LIN {X 0,Y 312.068,Z 552.76,A -85,B 0,C 180,E1 -16415.031,E2 -16415.031} C_VEL
LIN {X 0,Y 304.932,Z 536.125,A -85,B 0,C 180,E1 -16417.056,E2 -16417.056} C_VEL
LIN {X 0,Y 298.517,Z 522.21,A -85,B 0,C 180,E1 -16418.657,E2 -16418.657} C_VEL
LIN {X 0,Y 298.42,Z 521.626,A -85,B 0,C 180,E1 -16418.707,E2 -16418.707} C_VEL
LIN {X 0,Y 298.405,Z 521.628,A -85,B 0,C 180,E1 -16423.103,E2 -16423.103} C_VEL
LIN {X 0,Y 298.409,Z 521.626,A -85,B 0,C 180,E1 -16426.921,E2 -16426.921} C_VEL
LIN {X 0,Y 298.421,Z 521.626,A -85,B 0,C 180,E1 -16431.003,E2 -16431.003} C_VEL
LIN {X 0,Y 298.435,Z 521.723,A -85,B 0,C 180,E1 -16434.866,E2 -16434.866} C_VEL
LIN {X 0,Y 299.612,Z 527.188,A -85,B 0,C 180,E1 -16438.931,E2 -16438.931} C_VEL
LIN {X 0,Y 300.508,Z 532.409,A -85,B 0,C 180,E1 -16442.713,E2 -16442.713} C_VEL
LIN {X 0,Y 300.68,Z 534.35,A -85,B 0,C 180,E1 -16443.977,E2 -16443.977} C_VEL
LIN {X 0,Y 302.293,Z 537.797,A -85,B 0,C 180,E1 -16444.308,E2 -16444.308} C_VEL
LIN {X 0,Y 309.274,Z 552.419,A -85,B 0,C 180,E1 -16445.757,E2 -16445.757} C_VEL
LIN {X 0,Y 315.209,Z 567.429,A -85,B 0,C 180,E1 -16447.268,E2 -16447.268} C_VEL
LIN {X 0,Y 319.843,Z 581.754,A -85,B 0,C 180,E1 -16448.771,E2 -16448.771} C_VEL
LIN {X 0,Y 323.38,Z 594.422,A -85,B 0,C 180,E1 -16450.193,E2 -16450.193} C_VEL
LIN {X 0,Y 321.224,Z 608.572,A -85,B 0,C 180,E1 -16451.337,E2 -16451.337} C_VEL
LIN {X 0,Y 318.47,Z 623.738,A -85,B 0,C 180,E1 -16452.832,E2 -16452.832} C_VEL
LIN {X 0,Y 315.594,Z 637.637,A -85,B 0,C 180,E1 -16454.499,E2 -16454.499} C_VEL
LIN {X 0,Y 312.662,Z 650.484,A -85,B 0,C 180,E1 -16456.347,E2 -16456.347} C_VEL
LIN {X 0,Y 309.659,Z 663.096,A -85,B 0,C 180,E1 -16458.544,E2 -16458.544} C_VEL
LIN {X 0,Y 306.911,Z 673.805,A -85,B 0,C 180,E1 -16460.775,E2 -16460.775} C_VEL
LIN {X 0,Y 304.203,Z 684.215,A -85,B 0,C 180,E1 -16463.365,E2 -16463.365} C_VEL
LIN {X 0,Y 301.918,Z 692.982,A -85,B 0,C 180,E1 -16465.994,E2 -16465.994} C_VEL
LIN {X 0,Y 300.231,Z 700.324,A -85,B 0,C 180,E1 -16468.657,E2 -16468.657} C_VEL
LIN {X 0,Y 298.834,Z 706.332,A -85,B 0,C 180,E1 -16471.346,E2 -16471.346} C_VEL
LIN {X 0,Y 297.932,Z 711.223,A -85,B 0,C 180,E1 -16474.057,E2 -16474.057} C_VEL
LIN {X 0,Y 297.263,Z 715.069,A -85,B 0,C 180,E1 -16476.787,E2 -16476.787} C_VEL
LIN {X 0,Y 296.813,Z 717.858,A -85,B 0,C 180,E1 -16479.539,E2 -16479.539} C_VEL
LIN {X 0,Y 296.638,Z 719.722,A -85,B 0,C 180,E1 -16482.31,E2 -16482.31} C_VEL
LIN {X 0,Y 296.528,Z 720.531,A -85,B 0,C 180,E1 -16485.111,E2 -16485.111} C_VEL
LIN {X 0,Y 296.624,Z 720.427,A -85,B 0,C 180,E1 -16487.938,E2 -16487.938} C_VEL
LIN {X 0,Y 296.912,Z 719.249,A -85,B 0,C 180,E1 -16490.795,E2 -16490.795} C_VEL
LIN {X 0,Y 297.493,Z 717.043,A -85,B 0,C 180,E1 -16493.677,E2 -16493.677} C_VEL
LIN {X 0,Y 298.46,Z 713.748,A -85,B 0,C 180,E1 -16496.575,E2 -16496.575} C_VEL
LIN {X 0,Y 299.949,Z 708.491,A -85,B 0,C 180,E1 -16499.894,E2 -16499.894} C_VEL
LIN {X 0,Y 301.5,Z 703.345,A -85,B 0,C 180,E1 -16502.419,E2 -16502.419} C_VEL
LIN {X 0,Y 303.896,Z 696.084,A -85,B 0,C 180,E1 -16505.319,E2 -16505.319} C_VEL
LIN {X 0,Y 306.912,Z 687.177,A -85,B 0,C 180,E1 -16508.188,E2 -16508.188} C_VEL
LIN {X 0,Y 310.064,Z 677.773,A -85,B 0,C 180,E1 -16510.664,E2 -16510.664} C_VEL
LIN {X 0,Y 313.119,Z 668.301,A -85,B 0,C 180,E1 -16512.76,E2 -16512.76} C_VEL
LIN {X 0,Y 316.594,Z 657.264,A -85,B 0,C 180,E1 -16514.828,E2 -16514.828} C_VEL
LIN {X 0,Y 320.119,Z 645.238,A -85,B 0,C 180,E1 -16516.715,E2 -16516.715} C_VEL
LIN {X 0,Y 323.381,Z 632.92,A -85,B 0,C 180,E1 -16518.334,E2 -16518.334} C_VEL
LIN {X 0,Y 326.636,Z 619.578,A -85,B 0,C 180,E1 -16519.797,E2 -16519.797} C_VEL
LIN {X 0,Y 329.546,Z 605.586,A -85,B 0,C 180,E1 -16521.08,E2 -16521.08} C_VEL
LIN {X 0,Y 330.671,Z 599.403,A -85,B 0,C 180,E1 -16521.561,E2 -16521.561} C_VEL
LIN {X 0,Y 327.161,Z 585.978,A -85,B 0,C 180,E1 -16523.407,E2 -16523.407} C_VEL
LIN {X 0,Y 322.679,Z 573.581,A -85,B 0,C 180,E1 -16525.181,E2 -16525.181} C_VEL
LIN {X 0,Y 318.133,Z 563.085,A -85,B 0,C 180,E1 -16526.729,E2 -16526.729} C_VEL
LIN {X 0,Y 316.669,Z 560.38,A -85,B 0,C 180,E1 -16527.164,E2 -16527.164} C_VEL
LIN {X 0,Y 313.744,Z 557.363,A -85,B 0,C 180,E1 -16527.921,E2 -16527.921} C_VEL
LIN {X 0,Y 304.855,Z 551.294,A -85,B 0,C 180,E1 -16530.139,E2 -16530.139} C_VEL
LIN {X 0,Y 302.177,Z 547.886,A -85,B 0,C 180,E1 -16530.919,E2 -16530.919} C_VEL
LIN {X 0,Y 299.012,Z 543.525,A -85,B 0,C 180,E1 -16531.864,E2 -16531.864} C_VEL
LIN {X 0,Y 298.209,Z 542.203,A -85,B 0,C 180,E1 -16532.117,E2 -16532.117} C_VEL
LIN {X 0,Y 295.75,Z 539.263,A -85,B 0,C 180,E1 -16532.863,E2 -16532.863} C_VEL
LIN {X 0,Y 294.81,Z 537.165,A -85,B 0,C 180,E1 -16533.258,E2 -16533.258} C_VEL
LIN {X 0,Y 294.299,Z 534.199,A -85,B 0,C 180,E1 -16536.048,E2 -16536.048} C_VEL
LIN {X 0,Y 293.364,Z 529.878,A -85,B 0,C 180,E1 -16540.403,E2 -16540.403} C_VEL
LIN {X 0,Y 292.376,Z 525.78,A -85,B 0,C 180,E1 -16544.667,E2 -16544.667} C_VEL
LIN {X 0,Y 291.664,Z 523.407,A -85,B 0,C 180,E1 -16547.474,E2 -16547.474} C_VEL
LIN {X 0,Y 291.529,Z 522.475,A -85,B 0,C 180,E1 -16548.88,E2 -16548.88} C_VEL
LIN {X 0,Y 291.7,Z 522.453,A -85,B 0,C 180,E1 -16551.688,E2 -16551.688} C_VEL
LIN {X 0,Y 291.625,Z 522.464,A -85,B 0,C 180,E1 -16554.468,E2 -16554.468} C_VEL
LIN {X 0,Y 291.884,Z 522.428,A -85,B 0,C 180,E1 -16558.62,E2 -16558.62} C_VEL
LIN {X 0,Y 291.881,Z 522.429,A -85,B 0,C 180,E1 -16561.379,E2 -16561.379} C_VEL
LIN {X 0,Y 291.736,Z 522.455,A -85,B 0,C 180,E1 -16566.918,E2 -16566.918} C_VEL
LIN {X 0,Y 291.619,Z 522.46,A -85,B 0,C 180,E1 -16569.712,E2 -16569.712} C_VEL
LIN {X 0,Y 291.512,Z 522.483,A -85,B 0,C 180,E1 -16573.95,E2 -16573.95} C_VEL
LIN {X 0,Y 291.477,Z 522.439,A -85,B 0,C 180,E1 -16576.818,E2 -16576.818} C_VEL
LIN {X 0,Y 291.485,Z 522.46,A -85,B 0,C 180,E1 -16579.9,E2 -16579.9} C_VEL
LIN {X 0,Y 291.427,Z 522.446,A -85,B 0,C 180,E1 -16584.202,E2 -16584.202} C_VEL
LIN {X 0,Y 291.416,Z 522.525,A -85,B 0,C 180,E1 -16588.247,E2 -16588.247} C_VEL
LIN {X 0,Y 292.765,Z 528.915,A -85,B 0,C 180,E1 -16591.878,E2 -16591.878} C_VEL
LIN {X 0,Y 294.332,Z 536.056,A -85,B 0,C 180,E1 -16595.727,E2 -16595.727} C_VEL
LIN {X 0,Y 296.072,Z 544.172,A -85,B 0,C 180,E1 -16599.859,E2 -16599.859} C_VEL
LIN {X 0,Y 296.764,Z 547.425,A -85,B 0,C 180,E1 -16601.392,E2 -16601.392} C_VEL
LIN {X 0,Y 298.476,Z 553.641,A -85,B 0,C 180,E1 -16603.297,E2 -16603.297} C_VEL
LIN {X 0,Y 301.646,Z 559.124,A -85,B 0,C 180,E1 -16604.262,E2 -16604.262} C_VEL
LIN {X 0,Y 304.024,Z 563.851,A -85,B 0,C 180,E1 -16604.983,E2 -16604.983} C_VEL
LIN {X 0,Y 305.199,Z 565.983,A -85,B 0,C 180,E1 -16605.323,E2 -16605.323} C_VEL
LIN {X 0,Y 307.57,Z 571.571,A -85,B 0,C 180,E1 -16606.035,E2 -16606.035} C_VEL
LIN {X 0,Y 311.717,Z 584.767,A -85,B 0,C 180,E1 -16607.465,E2 -16607.465} C_VEL
LIN {X 0,Y 315.605,Z 601.039,A -85,B 0,C 180,E1 -16609.161,E2 -16609.161} C_VEL
LIN {X 0,Y 317.351,Z 612.191,A -85,B 0,C 180,E1 -16610.314,E2 -16610.314} C_VEL
LIN {X 0,Y 318.943,Z 628.691,A -85,B 0,C 180,E1 -16612.07,E2 -16612.07} C_VEL
LIN {X 0,Y 319.473,Z 641.632,A -85,B 0,C 180,E1 -16613.563,E2 -16613.563} C_VEL
LIN {X 0,Y 316.619,Z 654.375,A -85,B 0,C 180,E1 -16614.754,E2 -16614.754} C_VEL
LIN {X 0,Y 312.952,Z 668.352,A -85,B 0,C 180,E1 -16616.318,E2 -16616.318} C_VEL
LIN {X 0,Y 309.249,Z 681.452,A -85,B 0,C 180,E1 -16618.106,E2 -16618.106} C_VEL
LIN {X 0,Y 305.844,Z 693.144,A -85,B 0,C 180,E1 -16620.016,E2 -16620.016} C_VEL
LIN {X 0,Y 302.262,Z 704.878,A -85,B 0,C 180,E1 -16622.29,E2 -16622.29} C_VEL
LIN {X 0,Y 298.722,Z 716.22,A -85,B 0,C 180,E1 -16624.947,E2 -16624.947} C_VEL
LIN {X 0,Y 295.836,Z 725.738,A -85,B 0,C 180,E1 -16627.662,E2 -16627.662} C_VEL
LIN {X 0,Y 293.626,Z 733.778,A -85,B 0,C 180,E1 -16630.424,E2 -16630.424} C_VEL
LIN {X 0,Y 291.89,Z 740.531,A -85,B 0,C 180,E1 -16633.208,E2 -16633.208} C_VEL
LIN {X 0,Y 290.786,Z 746.03,A -85,B 0,C 180,E1 -16636.015,E2 -16636.015} C_VEL
LIN {X 0,Y 289.975,Z 750.428,A -85,B 0,C 180,E1 -16638.822,E2 -16638.822} C_VEL
LIN {X 0,Y 289.701,Z 753.787,A -85,B 0,C 180,E1 -16641.632,E2 -16641.632} C_VEL
LIN {X 0,Y 289.689,Z 756.102,A -85,B 0,C 180,E1 -16644.433,E2 -16644.433} C_VEL
LIN {X 0,Y 289.668,Z 757.442,A -85,B 0,C 180,E1 -16647.22,E2 -16647.22} C_VEL
LIN {X 0,Y 289.918,Z 757.758,A -85,B 0,C 180,E1 -16650.001,E2 -16650.001} C_VEL
LIN {X 0,Y 289.714,Z 757.082,A -85,B 0,C 180,E1 -16652.782,E2 -16652.782} C_VEL
LIN {X 0,Y 289.791,Z 754.905,A -85,B 0,C 180,E1 -16656.109,E2 -16656.109} C_VEL
LIN {X 0,Y 289.737,Z 752.618,A -85,B 0,C 180,E1 -16658.37,E2 -16658.37} C_VEL
LIN {X 0,Y 290.022,Z 748.721,A -85,B 0,C 180,E1 -16661.18,E2 -16661.18} C_VEL
LIN {X 0,Y 290.777,Z 743.764,A -85,B 0,C 180,E1 -16663.988,E2 -16663.988} C_VEL
LIN {X 0,Y 291.83,Z 737.527,A -85,B 0,C 180,E1 -16666.799,E2 -16666.799} C_VEL
LIN {X 0,Y 293.456,Z 729.927,A -85,B 0,C 180,E1 -16669.591,E2 -16669.591} C_VEL
LIN {X 0,Y 295.573,Z 720.817,A -85,B 0,C 180,E1 -16672.362,E2 -16672.362} C_VEL
LIN {X 0,Y 297.926,Z 711.447,A -85,B 0,C 180,E1 -16674.755,E2 -16674.755} C_VEL
LIN {X 0,Y 300.744,Z 701.517,A -85,B 0,C 180,E1 -16677.032,E2 -16677.032} C_VEL
LIN {X 0,Y 305.458,Z 687.681,A -85,B 0,C 180,E1 -16680.029,E2 -16680.029} C_VEL
LIN {X 0,Y 310.418,Z 674.005,A -85,B 0,C 180,E1 -16682.529,E2 -16682.529} C_VEL
LIN {X 0,Y 315.731,Z 659.951,A -85,B 0,C 180,E1 -16684.721,E2 -16684.721} C_VEL
LIN {X 0,Y 321.64,Z 644.618,A -85,B 0,C 180,E1 -16686.739,E2 -16686.739} C_VEL
LIN {X 0,Y 325.443,Z 627.689,A -85,B 0,C 180,E1 -16689.374,E2 -16689.374} C_VEL
LIN {X 0,Y 327.711,Z 618.124,A -85,B 0,C 180,E1 -16690.865,E2 -16690.865} C_VEL
LIN {X 0,Y 329.683,Z 608.688,A -85,B 0,C 180,E1 -16692.588,E2 -16692.588} C_VEL
LIN {X 0,Y 331.116,Z 602.16,A -85,B 0,C 180,E1 -16694.019,E2 -16694.019} C_VEL
LIN {X 0,Y 332.458,Z 596.698,A -85,B 0,C 180,E1 -16695.485,E2 -16695.485} C_VEL
LIN {X 0,Y 332.805,Z 595.493,A -85,B 0,C 180,E1 -16695.89,E2 -16695.89} C_VEL
LIN {X 0,Y 333.507,Z 593.023,A -85,B 0,C 180,E1 -16697.525,E2 -16697.525} C_VEL
LIN {X 0,Y 334.572,Z 592.021,A -85,B 0,C 180,E1 -16699.37,E2 -16699.37} C_VEL
LIN {X 0,Y 335.825,Z 592.61,A -85,B 0,C 180,E1 -16701.111,E2 -16701.111} C_VEL
LIN {X 0,Y 336.55,Z 593.309,A -85,B 0,C 180,E1 -16701.936,E2 -16701.936} C_VEL
LIN {X 0,Y 336.702,Z 594.466,A -85,B 0,C 180,E1 -16702.423,E2 -16702.423} C_VEL
LIN {X 0,Y 330.299,Z 609.275,A -85,B 0,C 180,E1 -16704.284,E2 -16704.284} C_VEL
LIN {X 0,Y 324.025,Z 623.317,A -85,B 0,C 180,E1 -16706.422,E2 -16706.422} C_VEL
LIN {X 0,Y 318.154,Z 636.055,A -85,B 0,C 180,E1 -16708.728,E2 -16708.728} C_VEL
LIN {X 0,Y 312.432,Z 648.32,A -85,B 0,C 180,E1 -16711.427,E2 -16711.427} C_VEL
LIN {X 0,Y 307.401,Z 658.917,A -85,B 0,C 180,E1 -16714.254,E2 -16714.254} C_VEL
LIN {X 0,Y 303.567,Z 666.914,A -85,B 0,C 180,E1 -16716.824,E2 -16716.824} C_VEL
LIN {X 0,Y 299.75,Z 674.929,A -85,B 0,C 180,E1 -16720.006,E2 -16720.006} C_VEL
LIN {X 0,Y 296.503,Z 681.705,A -85,B 0,C 180,E1 -16723.476,E2 -16723.476} C_VEL
LIN {X 0,Y 294.578,Z 685.761,A -85,B 0,C 180,E1 -16726.198,E2 -16726.198} C_VEL
LIN {X 0,Y 293.106,Z 688.796,A -85,B 0,C 180,E1 -16728.942,E2 -16728.942} C_VEL
LIN {X 0,Y 292.113,Z 690.843,A -85,B 0,C 180,E1 -16731.701,E2 -16731.701} C_VEL
LIN {X 0,Y 291.314,Z 691.996,A -85,B 0,C 180,E1 -16734.463,E2 -16734.463} C_VEL
LIN {X 0,Y 290.669,Z 692.161,A -85,B 0,C 180,E1 -16737.229,E2 -16737.229} C_VEL
LIN {X 0,Y 290.401,Z 691.421,A -85,B 0,C 180,E1 -16740.001,E2 -16740.001} C_VEL
LIN {X 0,Y 290.627,Z 689.591,A -85,B 0,C 180,E1 -16742.773,E2 -16742.773} C_VEL
LIN {X 0,Y 290.747,Z 686.851,A -85,B 0,C 180,E1 -16745.549,E2 -16745.549} C_VEL
LIN {X 0,Y 291.059,Z 683.042,A -85,B 0,C 180,E1 -16748.331,E2 -16748.331} C_VEL
LIN {X 0,Y 291.608,Z 678.11,A -85,B 0,C 180,E1 -16751.117,E2 -16751.117} C_VEL
LIN {X 0,Y 292.432,Z 672.021,A -85,B 0,C 180,E1 -16753.907,E2 -16753.907} C_VEL
LIN {X 0,Y 293.802,Z 664.583,A -85,B 0,C 180,E1 -16756.682,E2 -16756.682} C_VEL
LIN {X 0,Y 295.511,Z 655.655,A -85,B 0,C 180,E1 -16759.449,E2 -16759.449} C_VEL
LIN {X 0,Y 297.707,Z 645.056,A -85,B 0,C 180,E1 -16762.193,E2 -16762.193} C_VEL
LIN {X 0,Y 299.852,Z 634.147,A -85,B 0,C 180,E1 -16764.585,E2 -16764.585} C_VEL
LIN {X 0,Y 302.572,Z 621.424,A -85,B 0,C 180,E1 -16766.933,E2 -16766.933} C_VEL
LIN {X 0,Y 305.365,Z 607.68,A -85,B 0,C 180,E1 -16769.072,E2 -16769.072} C_VEL
LIN {X 0,Y 308.055,Z 593.873,A -85,B 0,C 180,E1 -16770.886,E2 -16770.886} C_VEL
LIN {X 0,Y 310.71,Z 579.23,A -85,B 0,C 180,E1 -16772.494,E2 -16772.494} C_VEL
LIN {X 0,Y 311.817,Z 571.97,A -85,B 0,C 180,E1 -16773.2,E2 -16773.2} C_VEL
LIN {X 0,Y 307.355,Z 559.617,A -85,B 0,C 180,E1 -16774.866,E2 -16774.866} C_VEL
LIN {X 0,Y 301.48,Z 545.18,A -85,B 0,C 180,E1 -16776.741,E2 -16776.741} C_VEL
LIN {X 0,Y 294.433,Z 529.331,A -85,B 0,C 180,E1 -16778.684,E2 -16778.684} C_VEL
LIN {X 0,Y 291.532,Z 523.367,A -85,B 0,C 180,E1 -16779.385,E2 -16779.385} C_VEL
LIN {X 0,Y 291.393,Z 522.501,A -85,B 0,C 180,E1 -16779.483,E2 -16779.483} C_VEL
LIN {X 0,Y 291.315,Z 522.51,A -85,B 0,C 180,E1 -16783.633,E2 -16783.633} C_VEL
LIN {X 0,Y 291.326,Z 522.511,A -85,B 0,C 180,E1 -16787.507,E2 -16787.507} C_VEL
LIN {X 0,Y 291.37,Z 522.505,A -85,B 0,C 180,E1 -16791.16,E2 -16791.16} C_VEL
LIN {X 0,Y 291.399,Z 522.611,A -85,B 0,C 180,E1 -16793.992,E2 -16793.992} C_VEL
LIN {X 0,Y 292.323,Z 526.946,A -85,B 0,C 180,E1 -16797.297,E2 -16797.297} C_VEL
LIN {X 0,Y 293.165,Z 531.342,A -85,B 0,C 180,E1 -16800.563,E2 -16800.563} C_VEL
LIN {X 0,Y 293.678,Z 534.633,A -85,B 0,C 180,E1 -16802.954,E2 -16802.954} C_VEL
LIN {X 0,Y 295.034,Z 537.774,A -85,B 0,C 180,E1 -16803.255,E2 -16803.255} C_VEL
LIN {X 0,Y 297.979,Z 543.093,A -85,B 0,C 180,E1 -16803.852,E2 -16803.852} C_VEL
LIN {X 0,Y 304.245,Z 556.889,A -85,B 0,C 180,E1 -16805.287,E2 -16805.287} C_VEL
LIN {X 0,Y 309.645,Z 570.83,A -85,B 0,C 180,E1 -16806.76,E2 -16806.76} C_VEL
LIN {X 0,Y 314.242,Z 585.645,A -85,B 0,C 180,E1 -16808.394,E2 -16808.394} C_VEL
LIN {X 0,Y 317.025,Z 595.953,A -85,B 0,C 180,E1 -16809.601,E2 -16809.601} C_VEL
LIN {X 0,Y 316.607,Z 600.05,A -85,B 0,C 180,E1 -16809.95,E2 -16809.95} C_VEL
LIN {X 0,Y 314.058,Z 614.736,A -85,B 0,C 180,E1 -16811.234,E2 -16811.234} C_VEL
LIN {X 0,Y 311.281,Z 628.973,A -85,B 0,C 180,E1 -16812.761,E2 -16812.761} C_VEL
LIN {X 0,Y 308.063,Z 643.223,A -85,B 0,C 180,E1 -16814.619,E2 -16814.619} C_VEL
LIN {X 0,Y 304.942,Z 656.155,A -85,B 0,C 180,E1 -16816.674,E2 -16816.674} C_VEL
LIN {X 0,Y 301.888,Z 667.985,A -85,B 0,C 180,E1 -16818.926,E2 -16818.926} C_VEL
LIN {X 0,Y 299.213,Z 678.09,A -85,B 0,C 180,E1 -16821.217,E2 -16821.217} C_VEL
LIN {X 0,Y 296.633,Z 687.902,A -85,B 0,C 180,E1 -16823.878,E2 -16823.878} C_VEL
LIN {X 0,Y 294.416,Z 696.158,A -85,B 0,C 180,E1 -16826.577,E2 -16826.577} C_VEL
LIN {X 0,Y 292.749,Z 702.969,A -85,B 0,C 180,E1 -16829.311,E2 -16829.311} C_VEL
LIN {X 0,Y 291.425,Z 708.624,A -85,B 0,C 180,E1 -16832.072,E2 -16832.072} C_VEL
LIN {X 0,Y 290.624,Z 713.137,A -85,B 0,C 180,E1 -16834.854,E2 -16834.854} C_VEL
LIN {X 0,Y 290.136,Z 715.861,A -85,B 0,C 180,E1 -16836.955,E2 -16836.955} C_VEL
LIN {X 0,Y 289.705,Z 718.53,A -85,B 0,C 180,E1 -16839.775,E2 -16839.775} C_VEL
LIN {X 0,Y 289.528,Z 720.286,A -85,B 0,C 180,E1 -16842.617,E2 -16842.617} C_VEL
LIN {X 0,Y 289.444,Z 721.023,A -85,B 0,C 180,E1 -16845.49,E2 -16845.49} C_VEL
LIN {X 0,Y 289.626,Z 720.652,A -85,B 0,C 180,E1 -16848.848,E2 -16848.848} C_VEL
LIN {X 0,Y 289.907,Z 719.555,A -85,B 0,C 180,E1 -16851.322,E2 -16851.322} C_VEL
LIN {X 0,Y 290.592,Z 717.214,A -85,B 0,C 180,E1 -16854.275,E2 -16854.275} C_VEL
LIN {X 0,Y 291.666,Z 713.805,A -85,B 0,C 180,E1 -16857.245,E2 -16857.245} C_VEL
LIN {X 0,Y 293.125,Z 708.984,A -85,B 0,C 180,E1 -16860.328,E2 -16860.328} C_VEL
LIN {X 0,Y 295.319,Z 702.313,A -85,B 0,C 180,E1 -16863.598,E2 -16863.598} C_VEL
LIN {X 0,Y 297.632,Z 695.728,A -85,B 0,C 180,E1 -16866.178,E2 -16866.178} C_VEL
LIN {X 0,Y 300.896,Z 686.635,A -85,B 0,C 180,E1 -16869.095,E2 -16869.095} C_VEL
LIN {X 0,Y 304.269,Z 677.111,A -85,B 0,C 180,E1 -16871.608,E2 -16871.608} C_VEL
LIN {X 0,Y 308.048,Z 665.732,A -85,B 0,C 180,E1 -16874.092,E2 -16874.092} C_VEL
LIN {X 0,Y 312.114,Z 653.156,A -85,B 0,C 180,E1 -16876.331,E2 -16876.331} C_VEL
LIN {X 0,Y 315.571,Z 641.406,A -85,B 0,C 180,E1 -16878.077,E2 -16878.077} C_VEL
LIN {X 0,Y 319.027,Z 628.425,A -85,B 0,C 180,E1 -16879.706,E2 -16879.706} C_VEL
LIN {X 0,Y 322.493,Z 613.913,A -85,B 0,C 180,E1 -16881.201,E2 -16881.201} C_VEL
LIN {X 0,Y 324.92,Z 602.182,A -85,B 0,C 180,E1 -16882.188,E2 -16882.188} C_VEL
LIN {X 0,Y 323.264,Z 594.426,A -85,B 0,C 180,E1 -16883.283,E2 -16883.283} C_VEL
LIN {X 0,Y 320.154,Z 583.941,A -85,B 0,C 180,E1 -16884.813,E2 -16884.813} C_VEL
LIN {X 0,Y 314.765,Z 570.031,A -85,B 0,C 180,E1 -16886.931,E2 -16886.931} C_VEL
LIN {X 0,Y 309.774,Z 560.044,A -85,B 0,C 180,E1 -16888.593,E2 -16888.593} C_VEL
LIN {X 0,Y 304.543,Z 551.551,A -85,B 0,C 180,E1 -16890.195,E2 -16890.195} C_VEL
LIN {X 0,Y 302.177,Z 547.886,A -85,B 0,C 180,E1 -16890.919,E2 -16890.919} C_VEL
LIN {X 0,Y 300.362,Z 545.843,A -85,B 0,C 180,E1 -16891.451,E2 -16891.451} C_VEL
LIN {X 0,Y 297.343,Z 544.559,A -85,B 0,C 180,E1 -16892.254,E2 -16892.254} C_VEL
LIN {X 0,Y 292.573,Z 543.398,A -85,B 0,C 180,E1 -16893.537,E2 -16893.537} C_VEL
LIN {X 0,Y 290.477,Z 542.015,A -85,B 0,C 180,E1 -16894.169,E2 -16894.169} C_VEL
LIN {X 0,Y 288.354,Z 539.004,A -85,B 0,C 180,E1 -16894.905,E2 -16894.905} C_VEL
LIN {X 0,Y 287.884,Z 537.831,A -85,B 0,C 180,E1 -16895.15,E2 -16895.15} C_VEL
LIN {X 0,Y 287.201,Z 534.564,A -85,B 0,C 180,E1 -16898.465,E2 -16898.465} C_VEL
LIN {X 0,Y 286.6,Z 531.729,A -85,B 0,C 180,E1 -16901.41,E2 -16901.41} C_VEL
LIN {X 0,Y 286.073,Z 529.219,A -85,B 0,C 180,E1 -16904.321,E2 -16904.321} C_VEL
LIN {X 0,Y 285.392,Z 526.753,A -85,B 0,C 180,E1 -16907.194,E2 -16907.194} C_VEL
LIN {X 0,Y 284.654,Z 523.331,A -85,B 0,C 180,E1 -16911.659,E2 -16911.659} C_VEL
LIN {X 0,Y 284.595,Z 523.34,A -85,B 0,C 180,E1 -16914.33,E2 -16914.33} C_VEL
LIN {X 0,Y 284.85,Z 523.304,A -85,B 0,C 180,E1 -16918.586,E2 -16918.586} C_VEL
LIN {X 0,Y 284.847,Z 523.305,A -85,B 0,C 180,E1 -16921.413,E2 -16921.413} C_VEL
LIN {X 0,Y 284.688,Z 523.334,A -85,B 0,C 180,E1 -16927.09,E2 -16927.09} C_VEL
LIN {X 0,Y 284.557,Z 523.342,A -85,B 0,C 180,E1 -16929.955,E2 -16929.955} C_VEL
LIN {X 0,Y 284.468,Z 523.362,A -85,B 0,C 180,E1 -16934.303,E2 -16934.303} C_VEL
LIN {X 0,Y 284.419,Z 523.314,A -85,B 0,C 180,E1 -16937.248,E2 -16937.248} C_VEL
LIN {X 0,Y 284.416,Z 523.348,A -85,B 0,C 180,E1 -16940.239,E2 -16940.239} C_VEL
LIN {X 0,Y 284.386,Z 523.324,A -85,B 0,C 180,E1 -16943.888,E2 -16943.888} C_VEL
LIN {X 0,Y 284.412,Z 523.547,A -85,B 0,C 180,E1 -16947.184,E2 -16947.184} C_VEL
LIN {X 0,Y 284.967,Z 526.134,A -85,B 0,C 180,E1 -16949.148,E2 -16949.148} C_VEL
LIN {X 0,Y 286.625,Z 533.849,A -85,B 0,C 180,E1 -16953.526,E2 -16953.526} C_VEL
LIN {X 0,Y 287.636,Z 538.467,A -85,B 0,C 180,E1 -16955.902,E2 -16955.902} C_VEL
LIN {X 0,Y 290.236,Z 548.399,A -85,B 0,C 180,E1 -16959.917,E2 -16959.917} C_VEL
LIN {X 0,Y 291.625,Z 553.109,A -85,B 0,C 180,E1 -16961.525,E2 -16961.525} C_VEL
LIN {X 0,Y 297.821,Z 563.754,A -85,B 0,C 180,E1 -16963.532,E2 -16963.532} C_VEL
LIN {X 0,Y 300.518,Z 569.122,A -85,B 0,C 180,E1 -16964.378,E2 -16964.378} C_VEL
LIN {X 0,Y 303.271,Z 575.471,A -85,B 0,C 180,E1 -16965.269,E2 -16965.269} C_VEL
LIN {X 0,Y 307.213,Z 588.978,A -85,B 0,C 180,E1 -16966.788,E2 -16966.788} C_VEL
LIN {X 0,Y 310.605,Z 604.754,A -85,B 0,C 180,E1 -16968.529,E2 -16968.529} C_VEL
LIN {X 0,Y 312.093,Z 615.786,A -85,B 0,C 180,E1 -16969.713,E2 -16969.713} C_VEL
LIN {X 0,Y 313.325,Z 632.527,A -85,B 0,C 180,E1 -16971.594,E2 -16971.594} C_VEL
LIN {X 0,Y 313.571,Z 643.992,A -85,B 0,C 180,E1 -16972.964,E2 -16972.964} C_VEL
LIN {X 0,Y 309.745,Z 659.026,A -85,B 0,C 180,E1 -16974.452,E2 -16974.452} C_VEL
LIN {X 0,Y 306.148,Z 671.945,A -85,B 0,C 180,E1 -16976.019,E2 -16976.019} C_VEL
LIN {X 0,Y 302.605,Z 683.749,A -85,B 0,C 180,E1 -16977.714,E2 -16977.714} C_VEL
LIN {X 0,Y 298.55,Z 696.753,A -85,B 0,C 180,E1 -16979.987,E2 -16979.987} C_VEL
LIN {X 0,Y 294.952,Z 707.814,A -85,B 0,C 180,E1 -16982.315,E2 -16982.315} C_VEL
LIN {X 0,Y 291.37,Z 718.597,A -85,B 0,C 180,E1 -16985.034,E2 -16985.034} C_VEL
LIN {X 0,Y 288.404,Z 728.142,A -85,B 0,C 180,E1 -16987.969,E2 -16987.969} C_VEL
LIN {X 0,Y 286.318,Z 735.393,A -85,B 0,C 180,E1 -16990.65,E2 -16990.65} C_VEL
LIN {X 0,Y 284.36,Z 743.165,A -85,B 0,C 180,E1 -16994.226,E2 -16994.226} C_VEL
LIN {X 0,Y 283.146,Z 749.132,A -85,B 0,C 180,E1 -16997.822,E2 -16997.822} C_VEL
LIN {X 0,Y 282.612,Z 753.42,A -85,B 0,C 180,E1 -17001.421,E2 -17001.421} C_VEL
LIN {X 0,Y 282.627,Z 755.697,A -85,B 0,C 180,E1 -17004.293,E2 -17004.293} C_VEL
LIN {X 0,Y 282.589,Z 757.018,A -85,B 0,C 180,E1 -17007.15,E2 -17007.15} C_VEL
LIN {X 0,Y 282.831,Z 757.297,A -85,B 0,C 180,E1 -17010.002,E2 -17010.002} C_VEL
LIN {X 0,Y 282.633,Z 756.603,A -85,B 0,C 180,E1 -17012.852,E2 -17012.852} C_VEL
LIN {X 0,Y 282.7,Z 754.545,A -85,B 0,C 180,E1 -17016.066,E2 -17016.066} C_VEL
LIN {X 0,Y 282.673,Z 752.074,A -85,B 0,C 180,E1 -17018.581,E2 -17018.581} C_VEL
LIN {X 0,Y 283.167,Z 747.036,A -85,B 0,C 180,E1 -17022.18,E2 -17022.18} C_VEL
LIN {X 0,Y 284.075,Z 741.298,A -85,B 0,C 180,E1 -17025.237,E2 -17025.237} C_VEL
LIN {X 0,Y 285.29,Z 735.068,A -85,B 0,C 180,E1 -17027.936,E2 -17027.936} C_VEL
LIN {X 0,Y 287.14,Z 727.116,A -85,B 0,C 180,E1 -17030.789,E2 -17030.789} C_VEL
LIN {X 0,Y 289.52,Z 717.506,A -85,B 0,C 180,E1 -17033.613,E2 -17033.613} C_VEL
LIN {X 0,Y 293.541,Z 704.191,A -85,B 0,C 180,E1 -17037.06,E2 -17037.06} C_VEL
LIN {X 0,Y 298.231,Z 691.414,A -85,B 0,C 180,E1 -17040.052,E2 -17040.052} C_VEL
LIN {X 0,Y 302.45,Z 680.274,A -85,B 0,C 180,E1 -17042.308,E2 -17042.308} C_VEL
LIN {X 0,Y 308.824,Z 664.602,A -85,B 0,C 180,E1 -17044.99,E2 -17044.99} C_VEL
LIN {X 0,Y 315.318,Z 649.165,A -85,B 0,C 180,E1 -17047.2,E2 -17047.2} C_VEL
LIN {X 0,Y 316.584,Z 645.955,A -85,B 0,C 180,E1 -17047.626,E2 -17047.626} C_VEL
LIN {X 0,Y 320.27,Z 632.107,A -85,B 0,C 180,E1 -17049.931,E2 -17049.931} C_VEL
LIN {X 0,Y 322.893,Z 623.265,A -85,B 0,C 180,E1 -17051.338,E2 -17051.338} C_VEL
LIN {X 0,Y 325.265,Z 614.413,A -85,B 0,C 180,E1 -17052.982,E2 -17052.982} C_VEL
LIN {X 0,Y 327.111,Z 607.79,A -85,B 0,C 180,E1 -17054.443,E2 -17054.443} C_VEL
LIN {X 0,Y 329.06,Z 601.713,A -85,B 0,C 180,E1 -17056.131,E2 -17056.131} C_VEL
LIN {X 0,Y 329.641,Z 600.043,A -85,B 0,C 180,E1 -17056.981,E2 -17056.981} C_VEL
LIN {X 0,Y 330.515,Z 598.415,A -85,B 0,C 180,E1 -17058.763,E2 -17058.763} C_VEL
LIN {X 0,Y 331.176,Z 598.203,A -85,B 0,C 180,E1 -17059.816,E2 -17059.816} C_VEL
LIN {X 0,Y 332.414,Z 598.97,A -85,B 0,C 180,E1 -17061.47,E2 -17061.47} C_VEL
LIN {X 0,Y 332.125,Z 600.055,A -85,B 0,C 180,E1 -17061.789,E2 -17061.789} C_VEL
LIN {X 0,Y 325.404,Z 614.025,A -85,B 0,C 180,E1 -17063.662,E2 -17063.662} C_VEL
LIN {X 0,Y 318.875,Z 627.305,A -85,B 0,C 180,E1 -17065.805,E2 -17065.805} C_VEL
LIN {X 0,Y 312.704,Z 639.419,A -85,B 0,C 180,E1 -17068.119,E2 -17068.119} C_VEL
LIN {X 0,Y 307.355,Z 649.865,A -85,B 0,C 180,E1 -17070.516,E2 -17070.516} C_VEL
LIN {X 0,Y 301.951,Z 660.274,A -85,B 0,C 180,E1 -17073.382,E2 -17073.382} C_VEL
LIN {X 0,Y 298.322,Z 667.254,A -85,B 0,C 180,E1 -17075.653,E2 -17075.653} C_VEL
LIN {X 0,Y 294.497,Z 674.593,A -85,B 0,C 180,E1 -17078.548,E2 -17078.548} C_VEL
LIN {X 0,Y 291.109,Z 680.996,A -85,B 0,C 180,E1 -17081.709,E2 -17081.709} C_VEL
LIN {X 0,Y 288.742,Z 685.357,A -85,B 0,C 180,E1 -17084.471,E2 -17084.471} C_VEL
LIN {X 0,Y 286.953,Z 688.77,A -85,B 0,C 180,E1 -17087.267,E2 -17087.267} C_VEL
LIN {X 0,Y 285.677,Z 691.143,A -85,B 0,C 180,E1 -17090.084,E2 -17090.084} C_VEL
LIN {X 0,Y 284.742,Z 692.613,A -85,B 0,C 180,E1 -17092.912,E2 -17092.912} C_VEL
LIN {X 0,Y 283.942,Z 693.167,A -85,B 0,C 180,E1 -17095.742,E2 -17095.742} C_VEL
LIN {X 0,Y 283.443,Z 692.754,A -85,B 0,C 180,E1 -17098.58,E2 -17098.58} C_VEL
LIN {X 0,Y 283.413,Z 691.382,A -85,B 0,C 180,E1 -17101.422,E2 -17101.422} C_VEL
LIN {X 0,Y 283.664,Z 688.964,A -85,B 0,C 180,E1 -17104.263,E2 -17104.263} C_VEL
LIN {X 0,Y 283.765,Z 685.618,A -85,B 0,C 180,E1 -17107.114,E2 -17107.114} C_VEL
LIN {X 0,Y 284.284,Z 681.126,A -85,B 0,C 180,E1 -17109.966,E2 -17109.966} C_VEL
LIN {X 0,Y 284.998,Z 675.492,A -85,B 0,C 180,E1 -17112.824,E2 -17112.824} C_VEL
LIN {X 0,Y 286.223,Z 668.641,A -85,B 0,C 180,E1 -17115.671,E2 -17115.671} C_VEL
LIN {X 0,Y 287.767,Z 660.354,A -85,B 0,C 180,E1 -17118.512,E2 -17118.512} C_VEL
LIN {X 0,Y 289.785,Z 650.444,A -85,B 0,C 180,E1 -17121.334,E2 -17121.334} C_VEL
LIN {X 0,Y 291.959,Z 640.048,A -85,B 0,C 180,E1 -17123.831,E2 -17123.831} C_VEL
LIN {X 0,Y 294.459,Z 628.427,A -85,B 0,C 180,E1 -17126.203,E2 -17126.203} C_VEL
LIN {X 0,Y 297.446,Z 614.837,A -85,B 0,C 180,E1 -17128.535,E2 -17128.535} C_VEL
LIN {X 0,Y 300.299,Z 600.567,A -85,B 0,C 180,E1 -17130.599,E2 -17130.599} C_VEL
LIN {X 0,Y 303.095,Z 585.518,A -85,B 0,C 180,E1 -17132.423,E2 -17132.423} C_VEL
LIN {X 0,Y 305.104,Z 574.353,A -85,B 0,C 180,E1 -17133.562,E2 -17133.562} C_VEL
LIN {X 0,Y 304.674,Z 572.116,A -85,B 0,C 180,E1 -17133.856,E2 -17133.856} C_VEL
LIN {X 0,Y 298.901,Z 556.7,A -85,B 0,C 180,E1 -17136.003,E2 -17136.003} C_VEL
LIN {X 0,Y 292.848,Z 542.251,A -85,B 0,C 180,E1 -17137.91,E2 -17137.91} C_VEL
LIN {X 0,Y 285.546,Z 526.543,A -85,B 0,C 180,E1 -17139.894,E2 -17139.894} C_VEL
LIN {X 0,Y 284.402,Z 523.965,A -85,B 0,C 180,E1 -17140.2,E2 -17140.2} C_VEL
LIN {X 0,Y 284.316,Z 523.382,A -85,B 0,C 180,E1 -17140.276,E2 -17140.276} C_VEL
LIN {X 0,Y 284.252,Z 523.391,A -85,B 0,C 180,E1 -17144.19,E2 -17144.19} C_VEL
LIN {X 0,Y 284.278,Z 523.387,A -85,B 0,C 180,E1 -17148.124,E2 -17148.124} C_VEL
LIN {X 0,Y 284.334,Z 523.38,A -85,B 0,C 180,E1 -17152.276,E2 -17152.276} C_VEL
LIN {X 0,Y 284.377,Z 523.432,A -85,B 0,C 180,E1 -17152.957,E2 -17152.957} C_VEL
LIN {X 0,Y 285.516,Z 528.891,A -85,B 0,C 180,E1 -17157.211,E2 -17157.211} C_VEL
LIN {X 0,Y 286.352,Z 533.346,A -85,B 0,C 180,E1 -17160.601,E2 -17160.601} C_VEL
LIN {X 0,Y 286.647,Z 535.066,A -85,B 0,C 180,E1 -17161.87,E2 -17161.87} C_VEL
LIN {X 0,Y 288.335,Z 538.532,A -85,B 0,C 180,E1 -17162.249,E2 -17162.249} C_VEL
LIN {X 0,Y 293.485,Z 548.231,A -85,B 0,C 180,E1 -17163.378,E2 -17163.378} C_VEL
LIN {X 0,Y 298.768,Z 560.113,A -85,B 0,C 180,E1 -17164.68,E2 -17164.68} C_VEL
LIN {X 0,Y 304.384,Z 575.242,A -85,B 0,C 180,E1 -17166.371,E2 -17166.371} C_VEL
LIN {X 0,Y 308.839,Z 590.348,A -85,B 0,C 180,E1 -17168.12,E2 -17168.12} C_VEL
LIN {X 0,Y 310.644,Z 597.311,A -85,B 0,C 180,E1 -17168.97,E2 -17168.97} C_VEL
LIN {X 0,Y 310.796,Z 599.159,A -85,B 0,C 180,E1 -17169.174,E2 -17169.174} C_VEL
LIN {X 0,Y 308.371,Z 612.914,A -85,B 0,C 180,E1 -17170.355,E2 -17170.355} C_VEL
LIN {X 0,Y 305.183,Z 628.802,A -85,B 0,C 180,E1 -17172.059,E2 -17172.059} C_VEL
LIN {X 0,Y 301.854,Z 643.131,A -85,B 0,C 180,E1 -17173.948,E2 -17173.948} C_VEL
LIN {X 0,Y 299.068,Z 654.273,A -85,B 0,C 180,E1 -17175.714,E2 -17175.714} C_VEL
LIN {X 0,Y 295.882,Z 666.475,A -85,B 0,C 180,E1 -17178.003,E2 -17178.003} C_VEL
LIN {X 0,Y 293.044,Z 676.907,A -85,B 0,C 180,E1 -17180.334,E2 -17180.334} C_VEL
LIN {X 0,Y 290.243,Z 686.966,A -85,B 0,C 180,E1 -17183.045,E2 -17183.045} C_VEL
LIN {X 0,Y 287.867,Z 695.404,A -85,B 0,C 180,E1 -17185.798,E2 -17185.798} C_VEL
LIN {X 0,Y 286.052,Z 702.459,A -85,B 0,C 180,E1 -17188.591,E2 -17188.591} C_VEL
LIN {X 0,Y 284.606,Z 708.325,A -85,B 0,C 180,E1 -17191.413,E2 -17191.413} C_VEL
LIN {X 0,Y 283.728,Z 712.945,A -85,B 0,C 180,E1 -17194.26,E2 -17194.26} C_VEL
LIN {X 0,Y 283.021,Z 716.599,A -85,B 0,C 180,E1 -17197.131,E2 -17197.131} C_VEL
LIN {X 0,Y 282.586,Z 719.206,A -85,B 0,C 180,E1 -17200.024,E2 -17200.024} C_VEL
LIN {X 0,Y 282.424,Z 720.837,A -85,B 0,C 180,E1 -17202.94,E2 -17202.94} C_VEL
LIN {X 0,Y 282.361,Z 721.516,A -85,B 0,C 180,E1 -17205.888,E2 -17205.888} C_VEL
LIN {X 0,Y 282.556,Z 721.103,A -85,B 0,C 180,E1 -17209.059,E2 -17209.059} C_VEL
LIN {X 0,Y 282.926,Z 719.854,A -85,B 0,C 180,E1 -17211.874,E2 -17211.874} C_VEL
LIN {X 0,Y 283.696,Z 717.39,A -85,B 0,C 180,E1 -17214.905,E2 -17214.905} C_VEL
LIN {X 0,Y 284.892,Z 713.844,A -85,B 0,C 180,E1 -17217.949,E2 -17217.949} C_VEL
LIN {X 0,Y 286.48,Z 709.108,A -85,B 0,C 180,E1 -17221.007,E2 -17221.007} C_VEL
LIN {X 0,Y 288.687,Z 702.801,A -85,B 0,C 180,E1 -17224.134,E2 -17224.134} C_VEL
LIN {X 0,Y 291.446,Z 695.375,A -85,B 0,C 180,E1 -17227.072,E2 -17227.072} C_VEL
LIN {X 0,Y 294.914,Z 686.104,A -85,B 0,C 180,E1 -17230.045,E2 -17230.045} C_VEL
LIN {X 0,Y 298.524,Z 676.385,A -85,B 0,C 180,E1 -17232.595,E2 -17232.595} C_VEL
LIN {X 0,Y 301.944,Z 666.595,A -85,B 0,C 180,E1 -17234.754,E2 -17234.754} C_VEL
LIN {X 0,Y 305.896,Z 654.85,A -85,B 0,C 180,E1 -17236.901,E2 -17236.901} C_VEL
LIN {X 0,Y 309.935,Z 641.815,A -85,B 0,C 180,E1 -17238.882,E2 -17238.882} C_VEL
LIN {X 0,Y 313.76,Z 628.129,A -85,B 0,C 180,E1 -17240.601,E2 -17240.601} C_VEL
LIN {X 0,Y 317.175,Z 614.203,A -85,B 0,C 180,E1 -17242.047,E2 -17242.047} C_VEL
LIN {X 0,Y 319.223,Z 604.78,A -85,B 0,C 180,E1 -17242.862,E2 -17242.862} C_VEL
LIN {X 0,Y 318.603,Z 600.599,A -85,B 0,C 180,E1 -17243.445,E2 -17243.445} C_VEL
LIN {X 0,Y 315.462,Z 588.77,A -85,B 0,C 180,E1 -17245.246,E2 -17245.246} C_VEL
LIN {X 0,Y 310.472,Z 575.022,A -85,B 0,C 180,E1 -17247.43,E2 -17247.43} C_VEL
LIN {X 0,Y 305.704,Z 564.973,A -85,B 0,C 180,E1 -17249.186,E2 -17249.186} C_VEL
LIN {X 0,Y 300.597,Z 556.408,A -85,B 0,C 180,E1 -17250.882,E2 -17250.882} C_VEL
LIN {X 0,Y 297.653,Z 552.006,A -85,B 0,C 180,E1 -17251.82,E2 -17251.82} C_VEL
LIN {X 0,Y 294.637,Z 547.539,A -85,B 0,C 180,E1 -17252.812,E2 -17252.812} C_VEL
LIN {X 0,Y 292.147,Z 544.044,A -85,B 0,C 180,E1 -17253.621,E2 -17253.621} C_VEL
LIN {X 0,Y 291.256,Z 542.763,A -85,B 0,C 180,E1 -17253.92,E2 -17253.92} C_VEL
LIN {X 0,Y 290.477,Z 542.015,A -85,B 0,C 180,E1 -17254.169,E2 -17254.169} C_VEL
LIN {X 0,Y 287.797,Z 540.141,A -85,B 0,C 180,E1 -17255.017,E2 -17255.017} C_VEL
LIN {X 0,Y 284.92,Z 539.194,A -85,B 0,C 180,E1 -17255.918,E2 -17255.918} C_VEL
LIN {X 0,Y 281.715,Z 538.474,A -85,B 0,C 180,E1 -17257.105,E2 -17257.105} C_VEL
LIN {X 0,Y 280.796,Z 537.89,A -85,B 0,C 180,E1 -17257.885,E2 -17257.885} C_VEL
LIN {X 0,Y 279.931,Z 533.755,A -85,B 0,C 180,E1 -17262.465,E2 -17262.465} C_VEL
LIN {X 0,Y 279.439,Z 531.317,A -85,B 0,C 180,E1 -17265.433,E2 -17265.433} C_VEL
LIN {X 0,Y 278.541,Z 527.94,A -85,B 0,C 180,E1 -17269.826,E2 -17269.826} C_VEL
LIN {X 0,Y 278.404,Z 526.837,A -85,B 0,C 180,E1 -17271.288,E2 -17271.288} C_VEL
LIN {X 0,Y 277.49,Z 524.225,A -85,B 0,C 180,E1 -17276.006,E2 -17276.006} C_VEL
LIN {X 0,Y 277.816,Z 524.18,A -85,B 0,C 180,E1 -17278.55,E2 -17278.55} C_VEL
LIN {X 0,Y 277.813,Z 524.18,A -85,B 0,C 180,E1 -17281.449,E2 -17281.449} C_VEL
LIN {X 0,Y 277.643,Z 524.211,A -85,B 0,C 180,E1 -17287.271,E2 -17287.271} C_VEL
LIN {X 0,Y 277.497,Z 524.224,A -85,B 0,C 180,E1 -17290.211,E2 -17290.211} C_VEL
LIN {X 0,Y 277.418,Z 524.232,A -85,B 0,C 180,E1 -17294.674,E2 -17294.674} C_VEL
LIN {X 0,Y 277.366,Z 524.202,A -85,B 0,C 180,E1 -17299.232,E2 -17299.232} C_VEL
LIN {X 0,Y 277.319,Z 524.364,A -85,B 0,C 180,E1 -17302.342,E2 -17302.342} C_VEL
LIN {X 0,Y 279.002,Z 528.014,A -85,B 0,C 180,E1 -17306.962,E2 -17306.962} C_VEL
LIN {X 0,Y 279.661,Z 531.279,A -85,B 0,C 180,E1 -17309.343,E2 -17309.343} C_VEL
LIN {X 0,Y 281.105,Z 538.229,A -85,B 0,C 180,E1 -17313.368,E2 -17313.368} C_VEL
LIN {X 0,Y 282.323,Z 543.234,A -85,B 0,C 180,E1 -17315.802,E2 -17315.802} C_VEL
LIN {X 0,Y 284.724,Z 552.51,A -85,B 0,C 180,E1 -17319.549,E2 -17319.549} C_VEL
LIN {X 0,Y 289.018,Z 559.768,A -85,B 0,C 180,E1 -17321.096,E2 -17321.096} C_VEL
LIN {X 0,Y 294.112,Z 568.558,A -85,B 0,C 180,E1 -17322.806,E2 -17322.806} C_VEL
LIN {X 0,Y 297.05,Z 574.526,A -85,B 0,C 180,E1 -17323.791,E2 -17323.791} C_VEL
LIN {X 0,Y 299.549,Z 580.966,A -85,B 0,C 180,E1 -17324.677,E2 -17324.677} C_VEL
LIN {X 0,Y 303.368,Z 596.137,A -85,B 0,C 180,E1 -17326.462,E2 -17326.462} C_VEL
LIN {X 0,Y 306.145,Z 611.762,A -85,B 0,C 180,E1 -17328.264,E2 -17328.264} C_VEL
LIN {X 0,Y 307.365,Z 627.398,A -85,B 0,C 180,E1 -17330.019,E2 -17330.019} C_VEL
LIN {X 0,Y 307.809,Z 643.013,A -85,B 0,C 180,E1 -17331.943,E2 -17331.943} C_VEL
LIN {X 0,Y 307.583,Z 646.197,A -85,B 0,C 180,E1 -17332.325,E2 -17332.325} C_VEL
LIN {X 0,Y 303.638,Z 660.842,A -85,B 0,C 180,E1 -17333.829,E2 -17333.829} C_VEL
LIN {X 0,Y 299.77,Z 673.969,A -85,B 0,C 180,E1 -17335.502,E2 -17335.502} C_VEL
LIN {X 0,Y 295.96,Z 685.839,A -85,B 0,C 180,E1 -17337.303,E2 -17337.303} C_VEL
LIN {X 0,Y 291.803,Z 698.479,A -85,B 0,C 180,E1 -17339.619,E2 -17339.619} C_VEL
LIN {X 0,Y 288.129,Z 709.286,A -85,B 0,C 180,E1 -17341.997,E2 -17341.997} C_VEL
LIN {X 0,Y 284.433,Z 719.728,A -85,B 0,C 180,E1 -17344.774,E2 -17344.774} C_VEL
LIN {X 0,Y 281.76,Z 727.783,A -85,B 0,C 180,E1 -17347.352,E2 -17347.352} C_VEL
LIN {X 0,Y 279.535,Z 735.178,A -85,B 0,C 180,E1 -17350.161,E2 -17350.161} C_VEL
LIN {X 0,Y 277.413,Z 742.884,A -85,B 0,C 180,E1 -17353.821,E2 -17353.821} C_VEL
LIN {X 0,Y 276.118,Z 748.805,A -85,B 0,C 180,E1 -17357.507,E2 -17357.507} C_VEL
LIN {X 0,Y 275.543,Z 753.056,A -85,B 0,C 180,E1 -17361.199,E2 -17361.199} C_VEL
LIN {X 0,Y 275.566,Z 755.294,A -85,B 0,C 180,E1 -17364.146,E2 -17364.146} C_VEL
LIN {X 0,Y 275.512,Z 756.596,A -85,B 0,C 180,E1 -17367.077,E2 -17367.077} C_VEL
LIN {X 0,Y 275.743,Z 756.834,A -85,B 0,C 180,E1 -17370.002,E2 -17370.002} C_VEL
LIN {X 0,Y 275.556,Z 756.12,A -85,B 0,C 180,E1 -17372.925,E2 -17372.925} C_VEL
LIN {X 0,Y 275.628,Z 754.149,A -85,B 0,C 180,E1 -17376.058,E2 -17376.058} C_VEL
LIN {X 0,Y 275.598,Z 751.512,A -85,B 0,C 180,E1 -17378.803,E2 -17378.803} C_VEL
LIN {X 0,Y 276.164,Z 746.432,A -85,B 0,C 180,E1 -17382.494,E2 -17382.494} C_VEL
LIN {X 0,Y 277.317,Z 739.512,A -85,B 0,C 180,E1 -17386.188,E2 -17386.188} C_VEL
LIN {X 0,Y 278.868,Z 732.513,A -85,B 0,C 180,E1 -17389.126,E2 -17389.126} C_VEL
LIN {X 0,Y 280.904,Z 724.061,A -85,B 0,C 180,E1 -17392.043,E2 -17392.043} C_VEL
LIN {X 0,Y 287.79,Z 702.876,A -85,B 0,C 180,E1 -17398.128,E2 -17398.128} C_VEL
LIN {X 0,Y 293.283,Z 689.116,A -85,B 0,C 180,E1 -17401.414,E2 -17401.414} C_VEL
LIN {X 0,Y 298.732,Z 676.357,A -85,B 0,C 180,E1 -17403.97,E2 -17403.97} C_VEL
LIN {X 0,Y 305.046,Z 662.202,A -85,B 0,C 180,E1 -17406.389,E2 -17406.389} C_VEL
LIN {X 0,Y 311.32,Z 648.555,A -85,B 0,C 180,E1 -17408.376,E2 -17408.376} C_VEL
LIN {X 0,Y 316.108,Z 633.468,A -85,B 0,C 180,E1 -17410.986,E2 -17410.986} C_VEL
LIN {X 0,Y 319.048,Z 625.019,A -85,B 0,C 180,E1 -17412.433,E2 -17412.433} C_VEL
LIN {X 0,Y 321.745,Z 617.004,A -85,B 0,C 180,E1 -17414.048,E2 -17414.048} C_VEL
LIN {X 0,Y 324.117,Z 610.331,A -85,B 0,C 180,E1 -17415.69,E2 -17415.69} C_VEL
LIN {X 0,Y 325.622,Z 606.827,A -85,B 0,C 180,E1 -17416.764,E2 -17416.764} C_VEL
LIN {X 0,Y 325.94,Z 606.099,A -85,B 0,C 180,E1 -17417.149,E2 -17417.149} C_VEL
LIN {X 0,Y 326.816,Z 604.495,A -85,B 0,C 180,E1 -17418.822,E2 -17418.822} C_VEL
LIN {X 0,Y 327.867,Z 604.394,A -85,B 0,C 180,E1 -17420.506,E2 -17420.506} C_VEL
LIN {X 0,Y 328.02,Z 604.92,A -85,B 0,C 180,E1 -17421.046,E2 -17421.046} C_VEL
LIN {X 0,Y 319.909,Z 620.213,A -85,B 0,C 180,E1 -17423.228,E2 -17423.228} C_VEL
LIN {X 0,Y 311.247,Z 635.888,A -85,B 0,C 180,E1 -17426.024,E2 -17426.024} C_VEL
LIN {X 0,Y 304.558,Z 647.821,A -85,B 0,C 180,E1 -17428.63,E2 -17428.63} C_VEL
LIN {X 0,Y 298.464,Z 658.636,A -85,B 0,C 180,E1 -17431.522,E2 -17431.522} C_VEL
LIN {X 0,Y 294.286,Z 665.804,A -85,B 0,C 180,E1 -17433.781,E2 -17433.781} C_VEL
LIN {X 0,Y 290.266,Z 672.9,A -85,B 0,C 180,E1 -17436.454,E2 -17436.454} C_VEL
LIN {X 0,Y 286.028,Z 680.212,A -85,B 0,C 180,E1 -17439.88,E2 -17439.88} C_VEL
LIN {X 0,Y 283.27,Z 684.929,A -85,B 0,C 180,E1 -17442.68,E2 -17442.68} C_VEL
LIN {X 0,Y 281.08,Z 688.594,A -85,B 0,C 180,E1 -17445.521,E2 -17445.521} C_VEL
LIN {X 0,Y 279.418,Z 691.392,A -85,B 0,C 180,E1 -17448.392,E2 -17448.392} C_VEL
LIN {X 0,Y 278.236,Z 693.134,A -85,B 0,C 180,E1 -17451.284,E2 -17451.284} C_VEL
LIN {X 0,Y 277.332,Z 694.045,A -85,B 0,C 180,E1 -17454.183,E2 -17454.183} C_VEL
LIN {X 0,Y 276.612,Z 693.978,A -85,B 0,C 180,E1 -17457.088,E2 -17457.088} C_VEL
LIN {X 0,Y 276.321,Z 692.972,A -85,B 0,C 180,E1 -17460.001,E2 -17460.001} C_VEL
LIN {X 0,Y 276.56,Z 690.963,A -85,B 0,C 180,E1 -17462.914,E2 -17462.914} C_VEL
LIN {X 0,Y 276.618,Z 687.966,A -85,B 0,C 180,E1 -17465.834,E2 -17465.834} C_VEL
LIN {X 0,Y 277.039,Z 683.964,A -85,B 0,C 180,E1 -17468.756,E2 -17468.756} C_VEL
LIN {X 0,Y 277.602,Z 678.77,A -85,B 0,C 180,E1 -17471.686,E2 -17471.686} C_VEL
LIN {X 0,Y 278.583,Z 672.388,A -85,B 0,C 180,E1 -17474.613,E2 -17474.613} C_VEL
LIN {X 0,Y 280.069,Z 664.689,A -85,B 0,C 180,E1 -17477.526,E2 -17477.526} C_VEL
LIN {X 0,Y 281.968,Z 655.5,A -85,B 0,C 180,E1 -17480.424,E2 -17480.424} C_VEL
LIN {X 0,Y 284.391,Z 644.564,A -85,B 0,C 180,E1 -17483.292,E2 -17483.292} C_VEL
LIN {X 0,Y 286.763,Z 633.283,A -85,B 0,C 180,E1 -17485.787,E2 -17485.787} C_VEL
LIN {X 0,Y 289.729,Z 620.113,A -85,B 0,C 180,E1 -17488.231,E2 -17488.231} C_VEL
LIN {X 0,Y 292.569,Z 606.92,A -85,B 0,C 180,E1 -17490.296,E2 -17490.296} C_VEL
LIN {X 0,Y 295.346,Z 592.83,A -85,B 0,C 180,E1 -17492.171,E2 -17492.171} C_VEL
LIN {X 0,Y 298.26,Z 577.582,A -85,B 0,C 180,E1 -17493.857,E2 -17493.857} C_VEL
LIN {X 0,Y 298.519,Z 576.006,A -85,B 0,C 180,E1 -17494.014,E2 -17494.014} C_VEL
LIN {X 0,Y 295.138,Z 566.078,A -85,B 0,C 180,E1 -17495.465,E2 -17495.465} C_VEL
LIN {X 0,Y 289.408,Z 551.555,A -85,B 0,C 180,E1 -17497.494,E2 -17497.494} C_VEL
LIN {X 0,Y 282.634,Z 536.121,A -85,B 0,C 180,E1 -17499.568,E2 -17499.568} C_VEL
LIN {X 0,Y 277.385,Z 525.044,A -85,B 0,C 180,E1 -17501.012,E2 -17501.012} C_VEL
LIN {X 0,Y 277.244,Z 524.264,A -85,B 0,C 180,E1 -17501.139,E2 -17501.139} C_VEL
LIN {X 0,Y 277.207,Z 524.267,A -85,B 0,C 180,E1 -17505.226,E2 -17505.226} C_VEL
LIN {X 0,Y 277.229,Z 524.265,A -85,B 0,C 180,E1 -17509.512,E2 -17509.512} C_VEL
LIN {X 0,Y 277.301,Z 524.305,A -85,B 0,C 180,E1 -17511.912,E2 -17511.912} C_VEL
LIN {X 0,Y 278.197,Z 528.576,A -85,B 0,C 180,E1 -17515.359,E2 -17515.359} C_VEL
LIN {X 0,Y 279.166,Z 533.072,A -85,B 0,C 180,E1 -17518.866,E2 -17518.866} C_VEL
LIN {X 0,Y 279.564,Z 535.468,A -85,B 0,C 180,E1 -17520.709,E2 -17520.709} C_VEL
LIN {X 0,Y 281.058,Z 538.667,A -85,B 0,C 180,E1 -17521.069,E2 -17521.069} C_VEL
LIN {X 0,Y 282.621,Z 541.171,A -85,B 0,C 180,E1 -17521.413,E2 -17521.413} C_VEL
LIN {X 0,Y 288.216,Z 551.598,A -85,B 0,C 180,E1 -17522.702,E2 -17522.702} C_VEL
LIN {X 0,Y 293.901,Z 564.917,A -85,B 0,C 180,E1 -17524.241,E2 -17524.241} C_VEL
LIN {X 0,Y 299.114,Z 579.719,A -85,B 0,C 180,E1 -17525.969,E2 -17525.969} C_VEL
LIN {X 0,Y 302.789,Z 592.768,A -85,B 0,C 180,E1 -17527.568,E2 -17527.568} C_VEL
LIN {X 0,Y 304.592,Z 600.64,A -85,B 0,C 180,E1 -17528.561,E2 -17528.561} C_VEL
LIN {X 0,Y 301.806,Z 615.666,A -85,B 0,C 180,E1 -17529.91,E2 -17529.91} C_VEL
LIN {X 0,Y 298.846,Z 629.904,A -85,B 0,C 180,E1 -17531.488,E2 -17531.488} C_VEL
LIN {X 0,Y 295.404,Z 644.165,A -85,B 0,C 180,E1 -17533.41,E2 -17533.41} C_VEL
LIN {X 0,Y 291.805,Z 658.045,A -85,B 0,C 180,E1 -17535.706,E2 -17535.706} C_VEL
LIN {X 0,Y 288.559,Z 669.71,A -85,B 0,C 180,E1 -17538.051,E2 -17538.051} C_VEL
LIN {X 0,Y 285.714,Z 679.677,A -85,B 0,C 180,E1 -17540.441,E2 -17540.441} C_VEL
LIN {X 0,Y 282.928,Z 689.38,A -85,B 0,C 180,E1 -17543.222,E2 -17543.222} C_VEL
LIN {X 0,Y 280.823,Z 696.604,A -85,B 0,C 180,E1 -17545.693,E2 -17545.693} C_VEL
LIN {X 0,Y 278.972,Z 703.51,A -85,B 0,C 180,E1 -17548.555,E2 -17548.555} C_VEL
LIN {X 0,Y 277.493,Z 709.25,A -85,B 0,C 180,E1 -17551.45,E2 -17551.45} C_VEL
LIN {X 0,Y 276.623,Z 713.798,A -85,B 0,C 180,E1 -17554.37,E2 -17554.37} C_VEL
LIN {X 0,Y 275.907,Z 717.328,A -85,B 0,C 180,E1 -17557.316,E2 -17557.316} C_VEL
LIN {X 0,Y 275.486,Z 719.877,A -85,B 0,C 180,E1 -17560.285,E2 -17560.285} C_VEL
LIN {X 0,Y 275.329,Z 721.655,A -85,B 0,C 180,E1 -17564.072,E2 -17564.072} C_VEL
LIN {X 0,Y 275.275,Z 722.005,A -85,B 0,C 180,E1 -17566.308,E2 -17566.308} C_VEL
LIN {X 0,Y 275.508,Z 721.531,A -85,B 0,C 180,E1 -17569.365,E2 -17569.365} C_VEL
LIN {X 0,Y 275.983,Z 720.102,A -85,B 0,C 180,E1 -17572.454,E2 -17572.454} C_VEL
LIN {X 0,Y 276.832,Z 717.57,A -85,B 0,C 180,E1 -17575.566,E2 -17575.566} C_VEL
LIN {X 0,Y 278.159,Z 713.885,A -85,B 0,C 180,E1 -17578.687,E2 -17578.687} C_VEL
LIN {X 0,Y 279.896,Z 709.018,A -85,B 0,C 180,E1 -17581.821,E2 -17581.821} C_VEL
LIN {X 0,Y 282.311,Z 702.793,A -85,B 0,C 180,E1 -17584.928,E2 -17584.928} C_VEL
LIN {X 0,Y 285.339,Z 695.04,A -85,B 0,C 180,E1 -17588.005,E2 -17588.005} C_VEL
LIN {X 0,Y 288.551,Z 686.867,A -85,B 0,C 180,E1 -17590.654,E2 -17590.654} C_VEL
LIN {X 0,Y 292.307,Z 677.21,A -85,B 0,C 180,E1 -17593.251,E2 -17593.251} C_VEL
LIN {X 0,Y 296.528,Z 665.719,A -85,B 0,C 180,E1 -17595.801,E2 -17595.801} C_VEL
LIN {X 0,Y 300.95,Z 653.011,A -85,B 0,C 180,E1 -17598.102,E2 -17598.102} C_VEL
LIN {X 0,Y 305.393,Z 638.962,A -85,B 0,C 180,E1 -17600.176,E2 -17600.176} C_VEL
LIN {X 0,Y 308.879,Z 626.588,A -85,B 0,C 180,E1 -17601.675,E2 -17601.675} C_VEL
LIN {X 0,Y 312.502,Z 611.875,A -85,B 0,C 180,E1 -17603.162,E2 -17603.162} C_VEL
LIN {X 0,Y 313.68,Z 606.187,A -85,B 0,C 180,E1 -17603.681,E2 -17603.681} C_VEL
LIN {X 0,Y 310.858,Z 594.122,A -85,B 0,C 180,E1 -17605.582,E2 -17605.582} C_VEL
LIN {X 0,Y 306.374,Z 580.631,A -85,B 0,C 180,E1 -17607.816,E2 -17607.816} C_VEL
LIN {X 0,Y 301.926,Z 570.513,A -85,B 0,C 180,E1 -17609.631,E2 -17609.631} C_VEL
LIN {X 0,Y 296.984,Z 561.799,A -85,B 0,C 180,E1 -17611.426,E2 -17611.426} C_VEL
LIN {X 0,Y 291.388,Z 553.132,A -85,B 0,C 180,E1 -17613.39,E2 -17613.39} C_VEL
LIN {X 0,Y 288.813,Z 549.213,A -85,B 0,C 180,E1 -17614.317,E2 -17614.317} C_VEL
LIN {X 0,Y 285.657,Z 545.209,A -85,B 0,C 180,E1 -17615.421,E2 -17615.421} C_VEL
LIN {X 0,Y 284.718,Z 543.723,A -85,B 0,C 180,E1 -17615.771,E2 -17615.771} C_VEL
LIN {X 0,Y 282.094,Z 540.831,A -85,B 0,C 180,E1 -17616.721,E2 -17616.721} C_VEL
LIN {X 0,Y 280.945,Z 538.495,A -85,B 0,C 180,E1 -17617.263,E2 -17617.263} C_VEL
LIN {X 0,Y 280.796,Z 537.89,A -85,B 0,C 180,E1 -17617.885,E2 -17617.885} C_VEL
LIN {X 0,Y 279.852,Z 537.118,A -85,B 0,C 180,E1 -17619.066,E2 -17619.066} C_VEL
LIN {X 0,Y 276.881,Z 536.564,A -85,B 0,C 180,E1 -17621.011,E2 -17621.011} C_VEL
LIN {X 0,Y 274.464,Z 536.232,A -85,B 0,C 180,E1 -17622.594,E2 -17622.594} C_VEL
LIN {X 0,Y 273.351,Z 535.682,A -85,B 0,C 180,E1 -17623.812,E2 -17623.812} C_VEL
LIN {X 0,Y 273.21,Z 535.36,A -85,B 0,C 180,E1 -17624.223,E2 -17624.223} C_VEL
LIN {X 0,Y 272.482,Z 532.116,A -85,B 0,C 180,E1 -17628.544,E2 -17628.544} C_VEL
LIN {X 0,Y 272.213,Z 530.463,A -85,B 0,C 180,E1 -17631.088,E2 -17631.088} C_VEL
LIN {X 0,Y 271.59,Z 528.682,A -85,B 0,C 180,E1 -17634.058,E2 -17634.058} C_VEL
LIN {X 0,Y 271.056,Z 526.375,A -85,B 0,C 180,E1 -17638.514,E2 -17638.514} C_VEL
LIN {X 0,Y 270.821,Z 525.381,A -85,B 0,C 180,E1 -17641.486,E2 -17641.486} C_VEL
LIN {X 0,Y 270.623,Z 525.08,A -85,B 0,C 180,E1 -17642.977,E2 -17642.977} C_VEL
LIN {X 0,Y 270.601,Z 525.085,A -85,B 0,C 180,E1 -17647.461,E2 -17647.461} C_VEL
LIN {X 0,Y 270.432,Z 525.107,A -85,B 0,C 180,E1 -17650.481,E2 -17650.481} C_VEL
LIN {X 0,Y 270.382,Z 525.182,A -85,B 0,C 180,E1 -17655.065,E2 -17655.065} C_VEL
LIN {X 0,Y 270.895,Z 527.147,A -85,B 0,C 180,E1 -17659.71,E2 -17659.71} C_VEL
LIN {X 0,Y 271.955,Z 529.281,A -85,B 0,C 180,E1 -17662.807,E2 -17662.807} C_VEL
LIN {X 0,Y 273.896,Z 533.553,A -85,B 0,C 180,E1 -17667.507,E2 -17667.507} C_VEL
LIN {X 0,Y 274.629,Z 537.2,A -85,B 0,C 180,E1 -17669.934,E2 -17669.934} C_VEL
LIN {X 0,Y 276.139,Z 544.486,A -85,B 0,C 180,E1 -17674.05,E2 -17674.05} C_VEL
LIN {X 0,Y 277.826,Z 551.764,A -85,B 0,C 180,E1 -17677.323,E2 -17677.323} C_VEL
LIN {X 0,Y 285.208,Z 563.967,A -85,B 0,C 180,E1 -17680.206,E2 -17680.206} C_VEL
LIN {X 0,Y 290.62,Z 573.876,A -85,B 0,C 180,E1 -17682.149,E2 -17682.149} C_VEL
LIN {X 0,Y 294.151,Z 581.614,A -85,B 0,C 180,E1 -17683.444,E2 -17683.444} C_VEL
LIN {X 0,Y 296.336,Z 589.214,A -85,B 0,C 180,E1 -17684.426,E2 -17684.426} C_VEL
LIN {X 0,Y 299.289,Z 603.496,A -85,B 0,C 180,E1 -17686.172,E2 -17686.172} C_VEL
LIN {X 0,Y 301.197,Z 616.903,A -85,B 0,C 180,E1 -17687.779,E2 -17687.779} C_VEL
LIN {X 0,Y 302.004,Z 633.044,A -85,B 0,C 180,E1 -17689.72,E2 -17689.72} C_VEL
LIN {X 0,Y 301.971,Z 646.8,A -85,B 0,C 180,E1 -17691.498,E2 -17691.498} C_VEL
LIN {X 0,Y 297.936,Z 661.247,A -85,B 0,C 180,E1 -17693.024,E2 -17693.024} C_VEL
LIN {X 0,Y 294.313,Z 673.019,A -85,B 0,C 180,E1 -17694.541,E2 -17694.541} C_VEL
LIN {X 0,Y 289.986,Z 686.001,A -85,B 0,C 180,E1 -17696.542,E2 -17696.542} C_VEL
LIN {X 0,Y 286.23,Z 696.901,A -85,B 0,C 180,E1 -17698.551,E2 -17698.551} C_VEL
LIN {X 0,Y 282.207,Z 708.057,A -85,B 0,C 180,E1 -17701.019,E2 -17701.019} C_VEL
LIN {X 0,Y 278.382,Z 718.412,A -85,B 0,C 180,E1 -17703.783,E2 -17703.783} C_VEL
LIN {X 0,Y 275.258,Z 727.282,A -85,B 0,C 180,E1 -17706.653,E2 -17706.653} C_VEL
LIN {X 0,Y 272.74,Z 734.95,A -85,B 0,C 180,E1 -17709.645,E2 -17709.645} C_VEL
LIN {X 0,Y 270.834,Z 741.188,A -85,B 0,C 180,E1 -17712.639,E2 -17712.639} C_VEL
LIN {X 0,Y 269.582,Z 746.302,A -85,B 0,C 180,E1 -17715.662,E2 -17715.662} C_VEL
LIN {X 0,Y 268.898,Z 749.406,A -85,B 0,C 180,E1 -17717.933,E2 -17717.933} C_VEL
LIN {X 0,Y 268.459,Z 752.695,A -85,B 0,C 180,E1 -17720.965,E2 -17720.965} C_VEL
LIN {X 0,Y 268.495,Z 754.939,A -85,B 0,C 180,E1 -17724.075,E2 -17724.075} C_VEL
LIN {X 0,Y 268.436,Z 756.17,A -85,B 0,C 180,E1 -17727,E2 -17727} C_VEL
LIN {X 0,Y 268.655,Z 756.372,A -85,B 0,C 180,E1 -17730.002,E2 -17730.002} C_VEL
LIN {X 0,Y 268.48,Z 755.631,A -85,B 0,C 180,E1 -17733.003,E2 -17733.003} C_VEL
LIN {X 0,Y 268.537,Z 753.782,A -85,B 0,C 180,E1 -17736.011,E2 -17736.011} C_VEL
LIN {X 0,Y 268.512,Z 750.94,A -85,B 0,C 180,E1 -17739.037,E2 -17739.037} C_VEL
LIN {X 0,Y 268.934,Z 746.945,A -85,B 0,C 180,E1 -17742.069,E2 -17742.069} C_VEL
LIN {X 0,Y 269.798,Z 741.829,A -85,B 0,C 180,E1 -17745.101,E2 -17745.101} C_VEL
LIN {X 0,Y 271.128,Z 735.505,A -85,B 0,C 180,E1 -17748.124,E2 -17748.124} C_VEL
LIN {X 0,Y 273.341,Z 726.694,A -85,B 0,C 180,E1 -17751.494,E2 -17751.494} C_VEL
LIN {X 0,Y 277.124,Z 714.205,A -85,B 0,C 180,E1 -17755.541,E2 -17755.541} C_VEL
LIN {X 0,Y 281.443,Z 703.429,A -85,B 0,C 180,E1 -17758.763,E2 -17758.763} C_VEL
LIN {X 0,Y 287.293,Z 689.959,A -85,B 0,C 180,E1 -17762.146,E2 -17762.146} C_VEL
LIN {X 0,Y 292.988,Z 677.745,A -85,B 0,C 180,E1 -17764.73,E2 -17764.73} C_VEL
LIN {X 0,Y 299.568,Z 664.21,A -85,B 0,C 180,E1 -17767.165,E2 -17767.165} C_VEL
LIN {X 0,Y 306.071,Z 651.144,A -85,B 0,C 180,E1 -17769.159,E2 -17769.159} C_VEL
LIN {X 0,Y 314.911,Z 628.429,A -85,B 0,C 180,E1 -17773.27,E2 -17773.27} C_VEL
LIN {X 0,Y 318.224,Z 620.173,A -85,B 0,C 180,E1 -17775.032,E2 -17775.032} C_VEL
LIN {X 0,Y 320.479,Z 615.126,A -85,B 0,C 180,E1 -17776.36,E2 -17776.36} C_VEL
LIN {X 0,Y 322.13,Z 611.88,A -85,B 0,C 180,E1 -17777.443,E2 -17777.443} C_VEL
LIN {X 0,Y 323.353,Z 610.304,A -85,B 0,C 180,E1 -17779.529,E2 -17779.529} C_VEL
LIN {X 0,Y 323.695,Z 610.219,A -85,B 0,C 180,E1 -17780.12,E2 -17780.12} C_VEL
LIN {X 0,Y 322.898,Z 611.869,A -85,B 0,C 180,E1 -17780.567,E2 -17780.567} C_VEL
LIN {X 0,Y 314.184,Z 626.525,A -85,B 0,C 180,E1 -17782.846,E2 -17782.846} C_VEL
LIN {X 0,Y 306.123,Z 639.834,A -85,B 0,C 180,E1 -17785.375,E2 -17785.375} C_VEL
LIN {X 0,Y 299.119,Z 651.109,A -85,B 0,C 180,E1 -17787.993,E2 -17787.993} C_VEL
LIN {X 0,Y 292.053,Z 662.448,A -85,B 0,C 180,E1 -17791.231,E2 -17791.231} C_VEL
LIN {X 0,Y 286.127,Z 671.789,A -85,B 0,C 180,E1 -17794.543,E2 -17794.543} C_VEL
LIN {X 0,Y 281.238,Z 679.453,A -85,B 0,C 180,E1 -17797.986,E2 -17797.986} C_VEL
LIN {X 0,Y 277.347,Z 685.519,A -85,B 0,C 180,E1 -17801.534,E2 -17801.534} C_VEL
LIN {X 0,Y 274.347,Z 690.081,A -85,B 0,C 180,E1 -17805.158,E2 -17805.158} C_VEL
LIN {X 0,Y 272.219,Z 693.147,A -85,B 0,C 180,E1 -17808.837,E2 -17808.837} C_VEL
LIN {X 0,Y 271.325,Z 694.306,A -85,B 0,C 180,E1 -17811.06,E2 -17811.06} C_VEL
LIN {X 0,Y 270.345,Z 695.047,A -85,B 0,C 180,E1 -17814.032,E2 -17814.032} C_VEL
LIN {X 0,Y 269.584,Z 694.895,A -85,B 0,C 180,E1 -17817.012,E2 -17817.012} C_VEL
LIN {X 0,Y 269.281,Z 693.728,A -85,B 0,C 180,E1 -17820.001,E2 -17820.001} C_VEL
LIN {X 0,Y 269.508,Z 691.634,A -85,B 0,C 180,E1 -17822.99,E2 -17822.99} C_VEL
LIN {X 0,Y 269.557,Z 688.498,A -85,B 0,C 180,E1 -17825.987,E2 -17825.987} C_VEL
LIN {X 0,Y 270.017,Z 684.344,A -85,B 0,C 180,E1 -17828.985,E2 -17828.985} C_VEL
LIN {X 0,Y 270.628,Z 679.072,A -85,B 0,C 180,E1 -17831.991,E2 -17831.991} C_VEL
LIN {X 0,Y 271.682,Z 672.528,A -85,B 0,C 180,E1 -17834.993,E2 -17834.993} C_VEL
LIN {X 0,Y 273.226,Z 664.663,A -85,B 0,C 180,E1 -17837.98,E2 -17837.98} C_VEL
LIN {X 0,Y 275.213,Z 655.279,A -85,B 0,C 180,E1 -17840.948,E2 -17840.948} C_VEL
LIN {X 0,Y 277.736,Z 644.142,A -85,B 0,C 180,E1 -17843.884,E2 -17843.884} C_VEL
LIN {X 0,Y 280.266,Z 632.711,A -85,B 0,C 180,E1 -17846.431,E2 -17846.431} C_VEL
LIN {X 0,Y 283.349,Z 619.326,A -85,B 0,C 180,E1 -17848.926,E2 -17848.926} C_VEL
LIN {X 0,Y 286.585,Z 604.719,A -85,B 0,C 180,E1 -17851.203,E2 -17851.203} C_VEL
LIN {X 0,Y 289.747,Z 588.728,A -85,B 0,C 180,E1 -17853.284,E2 -17853.284} C_VEL
LIN {X 0,Y 291.83,Z 578.338,A -85,B 0,C 180,E1 -17854.412,E2 -17854.412} C_VEL
LIN {X 0,Y 291.145,Z 575.306,A -85,B 0,C 180,E1 -17854.84,E2 -17854.84} C_VEL
LIN {X 0,Y 286.004,Z 561.373,A -85,B 0,C 180,E1 -17856.917,E2 -17856.917} C_VEL
LIN {X 0,Y 279.686,Z 545.978,A -85,B 0,C 180,E1 -17859.118,E2 -17859.118} C_VEL
LIN {X 0,Y 272.923,Z 531.477,A -85,B 0,C 180,E1 -17861.128,E2 -17861.128} C_VEL
LIN {X 0,Y 270.323,Z 525.994,A -85,B 0,C 180,E1 -17861.844,E2 -17861.844} C_VEL
LIN {X 0,Y 270.171,Z 525.143,A -85,B 0,C 180,E1 -17861.963,E2 -17861.963} C_VEL
LIN {X 0,Y 270.159,Z 525.145,A -85,B 0,C 180,E1 -17865.38,E2 -17865.38} C_VEL
LIN {X 0,Y 270.181,Z 525.144,A -85,B 0,C 180,E1 -17869.434,E2 -17869.434} C_VEL
LIN {X 0,Y 270.213,Z 525.168,A -85,B 0,C 180,E1 -17870.776,E2 -17870.776} C_VEL
LIN {X 0,Y 271.231,Z 529.581,A -85,B 0,C 180,E1 -17874.411,E2 -17874.411} C_VEL
LIN {X 0,Y 272.263,Z 534.561,A -85,B 0,C 180,E1 -17878.413,E2 -17878.413} C_VEL
LIN {X 0,Y 272.523,Z 536.066,A -85,B 0,C 180,E1 -17879.484,E2 -17879.484} C_VEL
LIN {X 0,Y 274.046,Z 539.194,A -85,B 0,C 180,E1 -17879.868,E2 -17879.868} C_VEL
LIN {X 0,Y 275.551,Z 541.511,A -85,B 0,C 180,E1 -17880.215,E2 -17880.215} C_VEL
LIN {X 0,Y 280.157,Z 549.61,A -85,B 0,C 180,E1 -17881.319,E2 -17881.319} C_VEL
LIN {X 0,Y 285.013,Z 559.655,A -85,B 0,C 180,E1 -17882.588,E2 -17882.588} C_VEL
LIN {X 0,Y 290.296,Z 573.319,A -85,B 0,C 180,E1 -17884.243,E2 -17884.243} C_VEL
LIN {X 0,Y 294.507,Z 586.586,A -85,B 0,C 180,E1 -17885.895,E2 -17885.895} C_VEL
LIN {X 0,Y 297.861,Z 599.887,A -85,B 0,C 180,E1 -17887.613,E2 -17887.613} C_VEL
LIN {X 0,Y 298.352,Z 602.686,A -85,B 0,C 180,E1 -17887.973,E2 -17887.973} C_VEL
LIN {X 0,Y 295.611,Z 616.842,A -85,B 0,C 180,E1 -17889.288,E2 -17889.288} C_VEL
LIN {X 0,Y 292.536,Z 630.957,A -85,B 0,C 180,E1 -17890.892,E2 -17890.892} C_VEL
LIN {X 0,Y 288.983,Z 645.144,A -85,B 0,C 180,E1 -17892.849,E2 -17892.849} C_VEL
LIN {X 0,Y 285.522,Z 658.013,A -85,B 0,C 180,E1 -17895.02,E2 -17895.02} C_VEL
LIN {X 0,Y 282.142,Z 669.765,A -85,B 0,C 180,E1 -17897.409,E2 -17897.409} C_VEL
LIN {X 0,Y 279.176,Z 679.803,A -85,B 0,C 180,E1 -17899.849,E2 -17899.849} C_VEL
LIN {X 0,Y 276.498,Z 688.81,A -85,B 0,C 180,E1 -17902.441,E2 -17902.441} C_VEL
LIN {X 0,Y 273.77,Z 697.802,A -85,B 0,C 180,E1 -17905.582,E2 -17905.582} C_VEL
LIN {X 0,Y 271.895,Z 704.562,A -85,B 0,C 180,E1 -17908.517,E2 -17908.517} C_VEL
LIN {X 0,Y 270.385,Z 710.166,A -85,B 0,C 180,E1 -17911.488,E2 -17911.488} C_VEL
LIN {X 0,Y 269.502,Z 714.653,A -85,B 0,C 180,E1 -17914.485,E2 -17914.485} C_VEL
LIN {X 0,Y 268.789,Z 718.056,A -85,B 0,C 180,E1 -17917.51,E2 -17917.51} C_VEL
LIN {X 0,Y 268.381,Z 720.533,A -85,B 0,C 180,E1 -17920.561,E2 -17920.561} C_VEL
LIN {X 0,Y 268.232,Z 722.124,A -85,B 0,C 180,E1 -17924.198,E2 -17924.198} C_VEL
LIN {X 0,Y 268.205,Z 722.442,A -85,B 0,C 180,E1 -17926.751,E2 -17926.751} C_VEL
LIN {X 0,Y 268.469,Z 721.904,A -85,B 0,C 180,E1 -17929.894,E2 -17929.894} C_VEL
LIN {X 0,Y 269.043,Z 720.347,A -85,B 0,C 180,E1 -17933.067,E2 -17933.067} C_VEL
LIN {X 0,Y 270.031,Z 717.752,A -85,B 0,C 180,E1 -17936.258,E2 -17936.258} C_VEL
LIN {X 0,Y 271.458,Z 713.933,A -85,B 0,C 180,E1 -17939.464,E2 -17939.464} C_VEL
LIN {X 0,Y 273.398,Z 708.924,A -85,B 0,C 180,E1 -17942.67,E2 -17942.67} C_VEL
LIN {X 0,Y 276.024,Z 702.592,A -85,B 0,C 180,E1 -17945.844,E2 -17945.844} C_VEL
LIN {X 0,Y 279.29,Z 694.705,A -85,B 0,C 180,E1 -17948.981,E2 -17948.981} C_VEL
LIN {X 0,Y 283.292,Z 685.078,A -85,B 0,C 180,E1 -17952.051,E2 -17952.051} C_VEL
LIN {X 0,Y 287.351,Z 674.933,A -85,B 0,C 180,E1 -17954.686,E2 -17954.686} C_VEL
LIN {X 0,Y 291.191,Z 664.901,A -85,B 0,C 180,E1 -17956.862,E2 -17956.862} C_VEL
LIN {X 0,Y 295.522,Z 652.936,A -85,B 0,C 180,E1 -17959.028,E2 -17959.028} C_VEL
LIN {X 0,Y 299.733,Z 640.043,A -85,B 0,C 180,E1 -17960.956,E2 -17960.956} C_VEL
LIN {X 0,Y 303.557,Z 627.051,A -85,B 0,C 180,E1 -17962.557,E2 -17962.557} C_VEL
LIN {X 0,Y 307.07,Z 613.356,A -85,B 0,C 180,E1 -17963.968,E2 -17963.968} C_VEL
LIN {X 0,Y 308.055,Z 609.102,A -85,B 0,C 180,E1 -17964.355,E2 -17964.355} C_VEL
LIN {X 0,Y 306.033,Z 598.736,A -85,B 0,C 180,E1 -17966.038,E2 -17966.038} C_VEL
LIN {X 0,Y 302.354,Z 586.712,A -85,B 0,C 180,E1 -17968.105,E2 -17968.105} C_VEL
LIN {X 0,Y 298.518,Z 577.119,A -85,B 0,C 180,E1 -17969.883,E2 -17969.883} C_VEL
LIN {X 0,Y 293.897,Z 568.042,A -85,B 0,C 180,E1 -17971.768,E2 -17971.768} C_VEL
LIN {X 0,Y 288.057,Z 558.635,A -85,B 0,C 180,E1 -17974.003,E2 -17974.003} C_VEL
LIN {X 0,Y 284.956,Z 554.105,A -85,B 0,C 180,E1 -17975.167,E2 -17975.167} C_VEL
LIN {X 0,Y 281.608,Z 549.395,A -85,B 0,C 180,E1 -17976.464,E2 -17976.464} C_VEL
LIN {X 0,Y 278.95,Z 545.996,A -85,B 0,C 180,E1 -17977.498,E2 -17977.498} C_VEL
LIN {X 0,Y 278.031,Z 544.518,A -85,B 0,C 180,E1 -17977.881,E2 -17977.881} C_VEL
LIN {X 0,Y 275.24,Z 541.609,A -85,B 0,C 180,E1 -17979.005,E2 -17979.005} C_VEL
LIN {X 0,Y 273.975,Z 539.161,A -85,B 0,C 180,E1 -17979.64,E2 -17979.64} C_VEL
LIN {X 0,Y 273.34,Z 535.89,A -85,B 0,C 180,E1 -17983.57,E2 -17983.57} C_VEL
LIN {X 0,Y 273.21,Z 535.36,A -85,B 0,C 180,E1 -17984.223,E2 -17984.223} C_VEL
LIN {X 0,Y 272.394,Z 534.715,A -85,B 0,C 180,E1 -17985.441,E2 -17985.441} C_VEL
LIN {X 0,Y 269.47,Z 534.554,A -85,B 0,C 180,E1 -17987.444,E2 -17987.444} C_VEL
LIN {X 0,Y 267.066,Z 534.568,A -85,B 0,C 180,E1 -17989.075,E2 -17989.075} C_VEL
LIN {X 0,Y 266.027,Z 534.263,A -85,B 0,C 180,E1 -17990.335,E2 -17990.335} C_VEL
LIN {X 0,Y 265.934,Z 533.996,A -85,B 0,C 180,E1 -17990.759,E2 -17990.759} C_VEL
LIN {X 0,Y 265.467,Z 532.284,A -85,B 0,C 180,E1 -17993.921,E2 -17993.921} C_VEL
LIN {X 0,Y 265.055,Z 530.142,A -85,B 0,C 180,E1 -17998.48,E2 -17998.48} C_VEL
LIN {X 0,Y 264.801,Z 529.143,A -85,B 0,C 180,E1 -18001.52,E2 -18001.52} C_VEL
LIN {X 0,Y 264.285,Z 528.42,A -85,B 0,C 180,E1 -18006.105,E2 -18006.105} C_VEL
LIN {X 0,Y 264.314,Z 528.44,A -85,B 0,C 180,E1 -18009.179,E2 -18009.179} C_VEL
LIN {X 0,Y 264.51,Z 529.112,A -85,B 0,C 180,E1 -18013.834,E2 -18013.834} C_VEL
LIN {X 0,Y 264.906,Z 530.359,A -85,B 0,C 180,E1 -18016.967,E2 -18016.967} C_VEL
LIN {X 0,Y 266.082,Z 532.989,A -85,B 0,C 180,E1 -18021.701,E2 -18021.701} C_VEL
LIN {X 0,Y 268.329,Z 537.77,A -85,B 0,C 180,E1 -18027.066,E2 -18027.066} C_VEL
LIN {X 0,Y 268.954,Z 540.33,A -85,B 0,C 180,E1 -18028.908,E2 -18028.908} C_VEL
LIN {X 0,Y 270.367,Z 547.462,A -85,B 0,C 180,E1 -18033.084,E2 -18033.084} C_VEL
LIN {X 0,Y 271.43,Z 551.583,A -85,B 0,C 180,E1 -18035.056,E2 -18035.056} C_VEL
LIN {X 0,Y 274.935,Z 557.393,A -85,B 0,C 180,E1 -18036.635,E2 -18036.635} C_VEL
LIN {X 0,Y 281.92,Z 569.042,A -85,B 0,C 180,E1 -18039.462,E2 -18039.462} C_VEL
LIN {X 0,Y 287.229,Z 579.345,A -85,B 0,C 180,E1 -18041.523,E2 -18041.523} C_VEL
LIN {X 0,Y 290.304,Z 586.689,A -85,B 0,C 180,E1 -18042.805,E2 -18042.805} C_VEL
LIN {X 0,Y 293.102,Z 598.631,A -85,B 0,C 180,E1 -18044.371,E2 -18044.371} C_VEL
LIN {X 0,Y 295.514,Z 614.63,A -85,B 0,C 180,E1 -18046.397,E2 -18046.397} C_VEL
LIN {X 0,Y 296.316,Z 627.324,A -85,B 0,C 180,E1 -18047.958,E2 -18047.958} C_VEL
LIN {X 0,Y 296.416,Z 643.3,A -85,B 0,C 180,E1 -18050.036,E2 -18050.036} C_VEL
LIN {X 0,Y 296.058,Z 648.961,A -85,B 0,C 180,E1 -18050.802,E2 -18050.802} C_VEL
LIN {X 0,Y 291.884,Z 662.925,A -85,B 0,C 180,E1 -18052.342,E2 -18052.342} C_VEL
LIN {X 0,Y 287.669,Z 675.982,A -85,B 0,C 180,E1 -18054.105,E2 -18054.105} C_VEL
LIN {X 0,Y 283.376,Z 688.125,A -85,B 0,C 180,E1 -18056.083,E2 -18056.083} C_VEL
LIN {X 0,Y 278.926,Z 700.22,A -85,B 0,C 180,E1 -18058.48,E2 -18058.48} C_VEL
LIN {X 0,Y 274.985,Z 710.591,A -85,B 0,C 180,E1 -18060.951,E2 -18060.951} C_VEL
LIN {X 0,Y 271.031,Z 720.717,A -85,B 0,C 180,E1 -18063.846,E2 -18063.846} C_VEL
LIN {X 0,Y 267.875,Z 729.26,A -85,B 0,C 180,E1 -18066.827,E2 -18066.827} C_VEL
LIN {X 0,Y 265.395,Z 736.374,A -85,B 0,C 180,E1 -18069.866,E2 -18069.866} C_VEL
LIN {X 0,Y 263.551,Z 742.319,A -85,B 0,C 180,E1 -18072.944,E2 -18072.944} C_VEL
LIN {X 0,Y 262.321,Z 747.093,A -85,B 0,C 180,E1 -18076.049,E2 -18076.049} C_VEL
LIN {X 0,Y 261.545,Z 750.816,A -85,B 0,C 180,E1 -18079.16,E2 -18079.16} C_VEL
LIN {X 0,Y 261.313,Z 753.526,A -85,B 0,C 180,E1 -18082.274,E2 -18082.274} C_VEL
LIN {X 0,Y 261.422,Z 754.639,A -85,B 0,C 180,E1 -18084.09,E2 -18084.09} C_VEL
LIN {X 0,Y 261.363,Z 755.737,A -85,B 0,C 180,E1 -18086.919,E2 -18086.919} C_VEL
LIN {X 0,Y 261.568,Z 755.909,A -85,B 0,C 180,E1 -18090.002,E2 -18090.002} C_VEL
LIN {X 0,Y 261.406,Z 755.128,A -85,B 0,C 180,E1 -18093.084,E2 -18093.084} C_VEL
LIN {X 0,Y 261.437,Z 753.249,A -85,B 0,C 180,E1 -18096.174,E2 -18096.174} C_VEL
LIN {X 0,Y 261.445,Z 750.358,A -85,B 0,C 180,E1 -18099.283,E2 -18099.283} C_VEL
LIN {X 0,Y 261.925,Z 746.338,A -85,B 0,C 180,E1 -18102.397,E2 -18102.397} C_VEL
LIN {X 0,Y 262.921,Z 740.647,A -85,B 0,C 180,E1 -18105.786,E2 -18105.786} C_VEL
LIN {X 0,Y 264.255,Z 734.801,A -85,B 0,C 180,E1 -18108.613,E2 -18108.613} C_VEL
LIN {X 0,Y 266.592,Z 726.007,A -85,B 0,C 180,E1 -18112.042,E2 -18112.042} C_VEL
LIN {X 0,Y 268.992,Z 718.504,A -85,B 0,C 180,E1 -18114.712,E2 -18114.712} C_VEL
LIN {X 0,Y 273.586,Z 707.599,A -85,B 0,C 180,E1 -18118.376,E2 -18118.376} C_VEL
LIN {X 0,Y 278.761,Z 696.356,A -85,B 0,C 180,E1 -18121.544,E2 -18121.544} C_VEL
LIN {X 0,Y 284.962,Z 683.732,A -85,B 0,C 180,E1 -18124.56,E2 -18124.56} C_VEL
LIN {X 0,Y 292.331,Z 669.65,A -85,B 0,C 180,E1 -18127.377,E2 -18127.377} C_VEL
LIN {X 0,Y 301.751,Z 652.152,A -85,B 0,C 180,E1 -18130.266,E2 -18130.266} C_VEL
LIN {X 0,Y 307.44,Z 639.035,A -85,B 0,C 180,E1 -18132.769,E2 -18132.769} C_VEL
LIN {X 0,Y 311.436,Z 630.59,A -85,B 0,C 180,E1 -18134.393,E2 -18134.393} C_VEL
LIN {X 0,Y 314.95,Z 623.373,A -85,B 0,C 180,E1 -18136.061,E2 -18136.061} C_VEL
LIN {X 0,Y 317.881,Z 617.999,A -85,B 0,C 180,E1 -18137.637,E2 -18137.637} C_VEL
LIN {X 0,Y 318.663,Z 616.762,A -85,B 0,C 180,E1 -18138.579,E2 -18138.579} C_VEL
LIN {X 0,Y 319.355,Z 616.211,A -85,B 0,C 180,E1 -18139.73,E2 -18139.73} C_VEL
LIN {X 0,Y 310.455,Z 629.793,A -85,B 0,C 180,E1 -18141.912,E2 -18141.912} C_VEL
LIN {X 0,Y 300.722,Z 644.152,A -85,B 0,C 180,E1 -18144.804,E2 -18144.804} C_VEL
LIN {X 0,Y 292.78,Z 655.849,A -85,B 0,C 180,E1 -18147.718,E2 -18147.718} C_VEL
LIN {X 0,Y 286.318,Z 665.237,A -85,B 0,C 180,E1 -18150.599,E2 -18150.599} C_VEL
LIN {X 0,Y 281.267,Z 672.488,A -85,B 0,C 180,E1 -18153.272,E2 -18153.272} C_VEL
LIN {X 0,Y 276.931,Z 678.751,A -85,B 0,C 180,E1 -18156.044,E2 -18156.044} C_VEL
LIN {X 0,Y 272.377,Z 685.144,A -85,B 0,C 180,E1 -18159.615,E2 -18159.615} C_VEL
LIN {X 0,Y 268.79,Z 690.055,A -85,B 0,C 180,E1 -18163.285,E2 -18163.285} C_VEL
LIN {X 0,Y 266.598,Z 692.881,A -85,B 0,C 180,E1 -18166.276,E2 -18166.276} C_VEL
LIN {X 0,Y 265.008,Z 694.849,A -85,B 0,C 180,E1 -18169.302,E2 -18169.302} C_VEL
LIN {X 0,Y 263.871,Z 695.872,A -85,B 0,C 180,E1 -18172.348,E2 -18172.348} C_VEL
LIN {X 0,Y 262.91,Z 696.04,A -85,B 0,C 180,E1 -18175.401,E2 -18175.401} C_VEL
LIN {X 0,Y 262.333,Z 695.256,A -85,B 0,C 180,E1 -18178.466,E2 -18178.466} C_VEL
LIN {X 0,Y 262.289,Z 693.481,A -85,B 0,C 180,E1 -18181.536,E2 -18181.536} C_VEL
LIN {X 0,Y 262.509,Z 690.772,A -85,B 0,C 180,E1 -18184.607,E2 -18184.607} C_VEL
LIN {X 0,Y 262.815,Z 686.086,A -85,B 0,C 180,E1 -18188.333,E2 -18188.333} C_VEL
LIN {X 0,Y 263.437,Z 680.744,A -85,B 0,C 180,E1 -18191.543,E2 -18191.543} C_VEL
LIN {X 0,Y 264.431,Z 674.406,A -85,B 0,C 180,E1 -18194.626,E2 -18194.626} C_VEL
LIN {X 0,Y 266.017,Z 666.498,A -85,B 0,C 180,E1 -18197.789,E2 -18197.789} C_VEL
LIN {X 0,Y 267.924,Z 657.625,A -85,B 0,C 180,E1 -18200.74,E2 -18200.74} C_VEL
LIN {X 0,Y 270.462,Z 646.737,A -85,B 0,C 180,E1 -18203.752,E2 -18203.752} C_VEL
LIN {X 0,Y 272.947,Z 635.537,A -85,B 0,C 180,E1 -18206.371,E2 -18206.371} C_VEL
LIN {X 0,Y 276.059,Z 622.507,A -85,B 0,C 180,E1 -18208.929,E2 -18208.929} C_VEL
LIN {X 0,Y 278.978,Z 609.639,A -85,B 0,C 180,E1 -18211.069,E2 -18211.069} C_VEL
LIN {X 0,Y 282.01,Z 595.686,A -85,B 0,C 180,E1 -18213.036,E2 -18213.036} C_VEL
LIN {X 0,Y 285,Z 581.057,A -85,B 0,C 180,E1 -18214.766,E2 -18214.766} C_VEL
LIN {X 0,Y 285.218,Z 579.391,A -85,B 0,C 180,E1 -18214.949,E2 -18214.949} C_VEL
LIN {X 0,Y 280.197,Z 565.309,A -85,B 0,C 180,E1 -18217.154,E2 -18217.154} C_VEL
LIN {X 0,Y 274.545,Z 551.207,A -85,B 0,C 180,E1 -18219.251,E2 -18219.251} C_VEL
LIN {X 0,Y 268.113,Z 537.013,A -85,B 0,C 180,E1 -18221.303,E2 -18221.303} C_VEL
LIN {X 0,Y 263.238,Z 526.649,A -85,B 0,C 180,E1 -18222.759,E2 -18222.759} C_VEL
LIN {X 0,Y 263.14,Z 526.021,A -85,B 0,C 180,E1 -18222.843,E2 -18222.843} C_VEL
LIN {X 0,Y 263.13,Z 526.022,A -85,B 0,C 180,E1 -18226.15,E2 -18226.15} C_VEL
LIN {X 0,Y 263.164,Z 526.207,A -85,B 0,C 180,E1 -18229.636,E2 -18229.636} C_VEL
LIN {X 0,Y 264.075,Z 530.089,A -85,B 0,C 180,E1 -18232.98,E2 -18232.98} C_VEL
LIN {X 0,Y 265.184,Z 535.025,A -85,B 0,C 180,E1 -18237.091,E2 -18237.091} C_VEL
LIN {X 0,Y 265.437,Z 536.404,A -85,B 0,C 180,E1 -18238.158,E2 -18238.158} C_VEL
LIN {X 0,Y 267.088,Z 539.726,A -85,B 0,C 180,E1 -18238.599,E2 -18238.599} C_VEL
LIN {X 0,Y 268.602,Z 542.098,A -85,B 0,C 180,E1 -18238.972,E2 -18238.972} C_VEL
LIN {X 0,Y 274.831,Z 552.686,A -85,B 0,C 180,E1 -18240.533,E2 -18240.533} C_VEL
LIN {X 0,Y 280.062,Z 563.905,A -85,B 0,C 180,E1 -18242.015,E2 -18242.015} C_VEL
LIN {X 0,Y 285.041,Z 577.416,A -85,B 0,C 180,E1 -18243.749,E2 -18243.749} C_VEL
LIN {X 0,Y 289.567,Z 592.697,A -85,B 0,C 180,E1 -18245.751,E2 -18245.751} C_VEL
LIN {X 0,Y 292.075,Z 603.569,A -85,B 0,C 180,E1 -18247.227,E2 -18247.227} C_VEL
LIN {X 0,Y 291.849,Z 606.209,A -85,B 0,C 180,E1 -18247.484,E2 -18247.484} C_VEL
LIN {X 0,Y 288.799,Z 621.054,A -85,B 0,C 180,E1 -18248.963,E2 -18248.963} C_VEL
LIN {X 0,Y 285.601,Z 634.515,A -85,B 0,C 180,E1 -18250.596,E2 -18250.596} C_VEL
LIN {X 0,Y 281.968,Z 648.18,A -85,B 0,C 180,E1 -18252.595,E2 -18252.595} C_VEL
LIN {X 0,Y 278.747,Z 659.82,A -85,B 0,C 180,E1 -18254.647,E2 -18254.647} C_VEL
LIN {X 0,Y 275.297,Z 671.39,A -85,B 0,C 180,E1 -18257.091,E2 -18257.091} C_VEL
LIN {X 0,Y 271.799,Z 682.556,A -85,B 0,C 180,E1 -18259.945,E2 -18259.945} C_VEL
LIN {X 0,Y 268.923,Z 691.919,A -85,B 0,C 180,E1 -18262.868,E2 -18262.868} C_VEL
LIN {X 0,Y 266.717,Z 698.92,A -85,B 0,C 180,E1 -18265.464,E2 -18265.464} C_VEL
LIN {X 0,Y 264.821,Z 705.604,A -85,B 0,C 180,E1 -18268.478,E2 -18268.478} C_VEL
LIN {X 0,Y 263.282,Z 711.076,A -85,B 0,C 180,E1 -18271.528,E2 -18271.528} C_VEL
LIN {X 0,Y 262.37,Z 715.484,A -85,B 0,C 180,E1 -18274.608,E2 -18274.608} C_VEL
LIN {X 0,Y 261.661,Z 718.785,A -85,B 0,C 180,E1 -18277.716,E2 -18277.716} C_VEL
LIN {X 0,Y 261.257,Z 721.142,A -85,B 0,C 180,E1 -18280.852,E2 -18280.852} C_VEL
LIN {X 0,Y 261.15,Z 722.595,A -85,B 0,C 180,E1 -18284.342,E2 -18284.342} C_VEL
LIN {X 0,Y 261.137,Z 722.874,A -85,B 0,C 180,E1 -18287.218,E2 -18287.218} C_VEL
LIN {X 0,Y 261.465,Z 722.278,A -85,B 0,C 180,E1 -18290.45,E2 -18290.45} C_VEL
LIN {X 0,Y 262.31,Z 720.162,A -85,B 0,C 180,E1 -18294.361,E2 -18294.361} C_VEL
LIN {X 0,Y 263.226,Z 717.897,A -85,B 0,C 180,E1 -18296.991,E2 -18296.991} C_VEL
LIN {X 0,Y 264.812,Z 713.985,A -85,B 0,C 180,E1 -18300.279,E2 -18300.279} C_VEL
LIN {X 0,Y 266.946,Z 708.831,A -85,B 0,C 180,E1 -18303.562,E2 -18303.562} C_VEL
LIN {X 0,Y 269.781,Z 702.346,A -85,B 0,C 180,E1 -18306.808,E2 -18306.808} C_VEL
LIN {X 0,Y 273.326,Z 694.345,A -85,B 0,C 180,E1 -18310,E2 -18310} C_VEL
LIN {X 0,Y 276.807,Z 686.364,A -85,B 0,C 180,E1 -18312.582,E2 -18312.582} C_VEL
LIN {X 0,Y 280.954,Z 676.572,A -85,B 0,C 180,E1 -18315.219,E2 -18315.219} C_VEL
LIN {X 0,Y 285.322,Z 665.725,A -85,B 0,C 180,E1 -18317.639,E2 -18317.639} C_VEL
LIN {X 0,Y 289.773,Z 653.965,A -85,B 0,C 180,E1 -18319.814,E2 -18319.814} C_VEL
LIN {X 0,Y 294.14,Z 641.105,A -85,B 0,C 180,E1 -18321.775,E2 -18321.775} C_VEL
LIN {X 0,Y 297.937,Z 628.853,A -85,B 0,C 180,E1 -18323.32,E2 -18323.32} C_VEL
LIN {X 0,Y 301.769,Z 614.604,A -85,B 0,C 180,E1 -18324.825,E2 -18324.825} C_VEL
LIN {X 0,Y 302.479,Z 611.652,A -85,B 0,C 180,E1 -18325.096,E2 -18325.096} C_VEL
LIN {X 0,Y 301.693,Z 606.117,A -85,B 0,C 180,E1 -18326.007,E2 -18326.007} C_VEL
LIN {X 0,Y 299.316,Z 596.566,A -85,B 0,C 180,E1 -18327.699,E2 -18327.699} C_VEL
LIN {X 0,Y 296.464,Z 587.522,A -85,B 0,C 180,E1 -18329.357,E2 -18329.357} C_VEL
LIN {X 0,Y 292.566,Z 578.237,A -85,B 0,C 180,E1 -18331.236,E2 -18331.236} C_VEL
LIN {X 0,Y 287.692,Z 569.17,A -85,B 0,C 180,E1 -18333.327,E2 -18333.327} C_VEL
LIN {X 0,Y 284.148,Z 563.428,A -85,B 0,C 180,E1 -18334.793,E2 -18334.793} C_VEL
LIN {X 0,Y 281.859,Z 559.822,A -85,B 0,C 180,E1 -18335.754,E2 -18335.754} C_VEL
LIN {X 0,Y 278.73,Z 555.327,A -85,B 0,C 180,E1 -18337.043,E2 -18337.043} C_VEL
LIN {X 0,Y 275.987,Z 551.429,A -85,B 0,C 180,E1 -18338.216,E2 -18338.216} C_VEL
LIN {X 0,Y 274.486,Z 549.76,A -85,B 0,C 180,E1 -18338.846,E2 -18338.846} C_VEL
LIN {X 0,Y 271.853,Z 546.115,A -85,B 0,C 180,E1 -18340.017,E2 -18340.017} C_VEL
LIN {X 0,Y 271.015,Z 545.096,A -85,B 0,C 180,E1 -18340.396,E2 -18340.396} C_VEL
LIN {X 0,Y 268.324,Z 542.249,A -85,B 0,C 180,E1 -18341.64,E2 -18341.64} C_VEL
LIN {X 0,Y 267.122,Z 539.974,A -85,B 0,C 180,E1 -18342.327,E2 -18342.327} C_VEL
LIN {X 0,Y 266.505,Z 536.977,A -85,B 0,C 180,E1 -18346.27,E2 -18346.27} C_VEL
LIN {X 0,Y 265.934,Z 533.996,A -85,B 0,C 180,E1 -18350.759,E2 -18350.759} C_VEL
LIN {X 0,Y 265.605,Z 533.634,A -85,B 0,C 180,E1 -18351.599,E2 -18351.599} C_VEL
LIN {X 0,Y 264.286,Z 533.595,A -85,B 0,C 180,E1 -18352.846,E2 -18352.846} C_VEL
LIN {X 0,Y 260.115,Z 534.359,A -85,B 0,C 180,E1 -18355.759,E2 -18355.759} C_VEL
LIN {X 0,Y 259.098,Z 534.357,A -85,B 0,C 180,E1 -18357.059,E2 -18357.059} C_VEL
LIN {X 0,Y 259.01,Z 534.231,A -85,B 0,C 180,E1 -18357.498,E2 -18357.498} C_VEL
LIN {X 0,Y 258.993,Z 533.41,A -85,B 0,C 180,E1 -18359.999,E2 -18359.999} C_VEL
LIN {X 0,Y 258.623,Z 532.69,A -85,B 0,C 180,E1 -18363.115,E2 -18363.115} C_VEL
LIN {X 0,Y 258.507,Z 532.449,A -85,B 0,C 180,E1 -18367.812,E2 -18367.812} C_VEL
LIN {X 0,Y 258.715,Z 533.141,A -85,B 0,C 180,E1 -18372.551,E2 -18372.551} C_VEL
LIN {X 0,Y 259.18,Z 534.141,A -85,B 0,C 180,E1 -18375.733,E2 -18375.733} C_VEL
LIN {X 0,Y 260.209,Z 536.761,A -85,B 0,C 180,E1 -18380.555,E2 -18380.555} C_VEL
LIN {X 0,Y 261.41,Z 539.394,A -85,B 0,C 180,E1 -18383.929,E2 -18383.929} C_VEL
LIN {X 0,Y 262.935,Z 542.39,A -85,B 0,C 180,E1 -18387.025,E2 -18387.025} C_VEL
LIN {X 0,Y 263.46,Z 544.717,A -85,B 0,C 180,E1 -18388.695,E2 -18388.695} C_VEL
LIN {X 0,Y 264.74,Z 550.913,A -85,B 0,C 180,E1 -18392.293,E2 -18392.293} C_VEL
LIN {X 0,Y 269.214,Z 558.195,A -85,B 0,C 180,E1 -18394.571,E2 -18394.571} C_VEL
LIN {X 0,Y 273.344,Z 565.268,A -85,B 0,C 180,E1 -18396.481,E2 -18396.481} C_VEL
LIN {X 0,Y 278.399,Z 573.786,A -85,B 0,C 180,E1 -18398.639,E2 -18398.639} C_VEL
LIN {X 0,Y 283.401,Z 584.096,A -85,B 0,C 180,E1 -18400.79,E2 -18400.79} C_VEL
LIN {X 0,Y 286.276,Z 591.374,A -85,B 0,C 180,E1 -18402.107,E2 -18402.107} C_VEL
LIN {X 0,Y 288.774,Z 604.377,A -85,B 0,C 180,E1 -18403.864,E2 -18403.864} C_VEL
LIN {X 0,Y 290.554,Z 618.483,A -85,B 0,C 180,E1 -18405.734,E2 -18405.734} C_VEL
LIN {X 0,Y 290.99,Z 631.811,A -85,B 0,C 180,E1 -18407.451,E2 -18407.451} C_VEL
LIN {X 0,Y 290.704,Z 646.617,A -85,B 0,C 180,E1 -18409.482,E2 -18409.482} C_VEL
LIN {X 0,Y 290.552,Z 649.632,A -85,B 0,C 180,E1 -18409.911,E2 -18409.911} C_VEL
LIN {X 0,Y 286.317,Z 663.371,A -85,B 0,C 180,E1 -18411.477,E2 -18411.477} C_VEL
LIN {X 0,Y 281.948,Z 676.254,A -85,B 0,C 180,E1 -18413.259,E2 -18413.259} C_VEL
LIN {X 0,Y 277.486,Z 688.316,A -85,B 0,C 180,E1 -18415.261,E2 -18415.261} C_VEL
LIN {X 0,Y 272.855,Z 700.302,A -85,B 0,C 180,E1 -18417.695,E2 -18417.695} C_VEL
LIN {X 0,Y 268.718,Z 710.58,A -85,B 0,C 180,E1 -18420.206,E2 -18420.206} C_VEL
LIN {X 0,Y 264.582,Z 720.621,A -85,B 0,C 180,E1 -18423.158,E2 -18423.158} C_VEL
LIN {X 0,Y 261.23,Z 729.113,A -85,B 0,C 180,E1 -18426.202,E2 -18426.202} C_VEL
LIN {X 0,Y 258.068,Z 737.785,A -85,B 0,C 180,E1 -18430.1,E2 -18430.1} C_VEL
LIN {X 0,Y 255.944,Z 744.59,A -85,B 0,C 180,E1 -18434.064,E2 -18434.064} C_VEL
LIN {X 0,Y 254.865,Z 748.748,A -85,B 0,C 180,E1 -18437.257,E2 -18437.257} C_VEL
LIN {X 0,Y 254.314,Z 751.953,A -85,B 0,C 180,E1 -18440.457,E2 -18440.457} C_VEL
LIN {X 0,Y 254.349,Z 754.34,A -85,B 0,C 180,E1 -18444.108,E2 -18444.108} C_VEL
LIN {X 0,Y 254.291,Z 755.296,A -85,B 0,C 180,E1 -18446.833,E2 -18446.833} C_VEL
LIN {X 0,Y 254.48,Z 755.446,A -85,B 0,C 180,E1 -18450.002,E2 -18450.002} C_VEL
LIN {X 0,Y 254.334,Z 754.62,A -85,B 0,C 180,E1 -18453.17,E2 -18453.17} C_VEL
LIN {X 0,Y 254.355,Z 752.716,A -85,B 0,C 180,E1 -18456.347,E2 -18456.347} C_VEL
LIN {X 0,Y 254.395,Z 749.776,A -85,B 0,C 180,E1 -18459.543,E2 -18459.543} C_VEL
LIN {X 0,Y 254.924,Z 745.732,A -85,B 0,C 180,E1 -18462.743,E2 -18462.743} C_VEL
LIN {X 0,Y 255.92,Z 740.355,A -85,B 0,C 180,E1 -18466.023,E2 -18466.023} C_VEL
LIN {X 0,Y 257.415,Z 734.076,A -85,B 0,C 180,E1 -18469.126,E2 -18469.126} C_VEL
LIN {X 0,Y 259.585,Z 726.235,A -85,B 0,C 180,E1 -18472.275,E2 -18472.275} C_VEL
LIN {X 0,Y 264.7,Z 713.496,A -85,B 0,C 180,E1 -18477.26,E2 -18477.26} C_VEL
LIN {X 0,Y 270.008,Z 702.549,A -85,B 0,C 180,E1 -18480.802,E2 -18480.802} C_VEL
LIN {X 0,Y 276.94,Z 689.272,A -85,B 0,C 180,E1 -18484.379,E2 -18484.379} C_VEL
LIN {X 0,Y 285.116,Z 674.728,A -85,B 0,C 180,E1 -18487.597,E2 -18487.597} C_VEL
LIN {X 0,Y 294.711,Z 658.447,A -85,B 0,C 180,E1 -18490.53,E2 -18490.53} C_VEL
LIN {X 0,Y 296.755,Z 654.952,A -85,B 0,C 180,E1 -18491.088,E2 -18491.088} C_VEL
LIN {X 0,Y 307.26,Z 634.632,A -85,B 0,C 180,E1 -18495.16,E2 -18495.16} C_VEL
LIN {X 0,Y 310.696,Z 628.507,A -85,B 0,C 180,E1 -18496.613,E2 -18496.613} C_VEL
LIN {X 0,Y 313.181,Z 624.435,A -85,B 0,C 180,E1 -18497.779,E2 -18497.779} C_VEL
LIN {X 0,Y 314.185,Z 622.986,A -85,B 0,C 180,E1 -18498.382,E2 -18498.382} C_VEL
LIN {X 0,Y 314.577,Z 622.427,A -85,B 0,C 180,E1 -18498.819,E2 -18498.819} C_VEL
LIN {X 0,Y 313.348,Z 624.243,A -85,B 0,C 180,E1 -18499.426,E2 -18499.426} C_VEL
LIN {X 0,Y 303.814,Z 637.305,A -85,B 0,C 180,E1 -18501.772,E2 -18501.772} C_VEL
LIN {X 0,Y 295.142,Z 648.978,A -85,B 0,C 180,E1 -18504.311,E2 -18504.311} C_VEL
LIN {X 0,Y 288.092,Z 658.303,A -85,B 0,C 180,E1 -18506.789,E2 -18506.789} C_VEL
LIN {X 0,Y 280.67,Z 668.098,A -85,B 0,C 180,E1 -18509.948,E2 -18509.948} C_VEL
LIN {X 0,Y 274.134,Z 676.587,A -85,B 0,C 180,E1 -18513.344,E2 -18513.344} C_VEL
LIN {X 0,Y 268.701,Z 683.541,A -85,B 0,C 180,E1 -18516.901,E2 -18516.901} C_VEL
LIN {X 0,Y 265.137,Z 688.007,A -85,B 0,C 180,E1 -18519.844,E2 -18519.844} C_VEL
LIN {X 0,Y 262.168,Z 691.606,A -85,B 0,C 180,E1 -18522.85,E2 -18522.85} C_VEL
LIN {X 0,Y 259.84,Z 694.299,A -85,B 0,C 180,E1 -18525.912,E2 -18525.912} C_VEL
LIN {X 0,Y 258.124,Z 696.077,A -85,B 0,C 180,E1 -18529.013,E2 -18529.013} C_VEL
LIN {X 0,Y 256.921,Z 696.971,A -85,B 0,C 180,E1 -18532.14,E2 -18532.14} C_VEL
LIN {X 0,Y 255.902,Z 696.974,A -85,B 0,C 180,E1 -18535.275,E2 -18535.275} C_VEL
LIN {X 0,Y 255.297,Z 696.082,A -85,B 0,C 180,E1 -18538.423,E2 -18538.423} C_VEL
LIN {X 0,Y 255.223,Z 694.147,A -85,B 0,C 180,E1 -18541.579,E2 -18541.579} C_VEL
LIN {X 0,Y 255.46,Z 691.305,A -85,B 0,C 180,E1 -18544.735,E2 -18544.735} C_VEL
LIN {X 0,Y 255.766,Z 686.698,A -85,B 0,C 180,E1 -18548.415,E2 -18548.415} C_VEL
LIN {X 0,Y 256.445,Z 680.992,A -85,B 0,C 180,E1 -18551.862,E2 -18551.862} C_VEL
LIN {X 0,Y 257.501,Z 674.482,A -85,B 0,C 180,E1 -18555.028,E2 -18555.028} C_VEL
LIN {X 0,Y 259.201,Z 666.106,A -85,B 0,C 180,E1 -18558.376,E2 -18558.376} C_VEL
LIN {X 0,Y 261.488,Z 656.025,A -85,B 0,C 180,E1 -18561.689,E2 -18561.689} C_VEL
LIN {X 0,Y 263.851,Z 646.289,A -85,B 0,C 180,E1 -18564.385,E2 -18564.385} C_VEL
LIN {X 0,Y 266.483,Z 634.914,A -85,B 0,C 180,E1 -18567.062,E2 -18567.062} C_VEL
LIN {X 0,Y 269.721,Z 621.672,A -85,B 0,C 180,E1 -18569.675,E2 -18569.675} C_VEL
LIN {X 0,Y 272.956,Z 607.873,A -85,B 0,C 180,E1 -18571.956,E2 -18571.956} C_VEL
LIN {X 0,Y 275.869,Z 594.227,A -85,B 0,C 180,E1 -18573.869,E2 -18573.869} C_VEL
LIN {X 0,Y 278.363,Z 582.45,A -85,B 0,C 180,E1 -18575.278,E2 -18575.278} C_VEL
LIN {X 0,Y 278.427,Z 580.775,A -85,B 0,C 180,E1 -18575.491,E2 -18575.491} C_VEL
LIN {X 0,Y 273.693,Z 567.585,A -85,B 0,C 180,E1 -18577.632,E2 -18577.632} C_VEL
LIN {X 0,Y 267.609,Z 552.291,A -85,B 0,C 180,E1 -18579.987,E2 -18579.987} C_VEL
LIN {X 0,Y 260.449,Z 536.476,A -85,B 0,C 180,E1 -18582.382,E2 -18582.382} C_VEL
LIN {X 0,Y 256.194,Z 527.593,A -85,B 0,C 180,E1 -18583.669,E2 -18583.669} C_VEL
LIN {X 0,Y 256.074,Z 526.899,A -85,B 0,C 180,E1 -18583.77,E2 -18583.77} C_VEL
LIN {X 0,Y 256.098,Z 526.97,A -85,B 0,C 180,E1 -18588.182,E2 -18588.182} C_VEL
LIN {X 0,Y 257.212,Z 531.744,A -85,B 0,C 180,E1 -18592.411,E2 -18592.411} C_VEL
LIN {X 0,Y 258.237,Z 536.483,A -85,B 0,C 180,E1 -18596.456,E2 -18596.456} C_VEL
LIN {X 0,Y 258.393,Z 537.028,A -85,B 0,C 180,E1 -18596.753,E2 -18596.753} C_VEL
LIN {X 0,Y 260.271,Z 540.429,A -85,B 0,C 180,E1 -18597.271,E2 -18597.271} C_VEL
LIN {X 0,Y 261.47,Z 542.153,A -85,B 0,C 180,E1 -18597.581,E2 -18597.581} C_VEL
LIN {X 0,Y 269.398,Z 555.741,A -85,B 0,C 180,E1 -18599.695,E2 -18599.695} C_VEL
LIN {X 0,Y 274.638,Z 567.025,A -85,B 0,C 180,E1 -18601.303,E2 -18601.303} C_VEL
LIN {X 0,Y 279.388,Z 580.253,A -85,B 0,C 180,E1 -18603.076,E2 -18603.076} C_VEL
LIN {X 0,Y 283.562,Z 594.851,A -85,B 0,C 180,E1 -18605.079,E2 -18605.079} C_VEL
LIN {X 0,Y 286.039,Z 606.02,A -85,B 0,C 180,E1 -18606.656,E2 -18606.656} C_VEL
LIN {X 0,Y 282.964,Z 620.67,A -85,B 0,C 180,E1 -18608.125,E2 -18608.125} C_VEL
LIN {X 0,Y 279.683,Z 634.275,A -85,B 0,C 180,E1 -18609.785,E2 -18609.785} C_VEL
LIN {X 0,Y 275.919,Z 648.065,A -85,B 0,C 180,E1 -18611.817,E2 -18611.817} C_VEL
LIN {X 0,Y 272.527,Z 659.811,A -85,B 0,C 180,E1 -18613.904,E2 -18613.904} C_VEL
LIN {X 0,Y 268.934,Z 671.432,A -85,B 0,C 180,E1 -18616.395,E2 -18616.395} C_VEL
LIN {X 0,Y 265.748,Z 681.349,A -85,B 0,C 180,E1 -18618.944,E2 -18618.944} C_VEL
LIN {X 0,Y 262.669,Z 690.893,A -85,B 0,C 180,E1 -18621.885,E2 -18621.885} C_VEL
LIN {X 0,Y 260.257,Z 698.208,A -85,B 0,C 180,E1 -18624.575,E2 -18624.575} C_VEL
LIN {X 0,Y 258.174,Z 705.065,A -85,B 0,C 180,E1 -18627.658,E2 -18627.658} C_VEL
LIN {X 0,Y 256.511,Z 710.759,A -85,B 0,C 180,E1 -18630.783,E2 -18630.783} C_VEL
LIN {X 0,Y 255.477,Z 715.294,A -85,B 0,C 180,E1 -18633.942,E2 -18633.942} C_VEL
LIN {X 0,Y 254.77,Z 718.42,A -85,B 0,C 180,E1 -18636.736,E2 -18636.736} C_VEL
LIN {X 0,Y 254.326,Z 720.739,A -85,B 0,C 180,E1 -18639.542,E2 -18639.542} C_VEL
LIN {X 0,Y 254.101,Z 722.527,A -85,B 0,C 180,E1 -18642.782,E2 -18642.782} C_VEL
LIN {X 0,Y 254.034,Z 723.288,A -85,B 0,C 180,E1 -18646.059,E2 -18646.059} C_VEL
LIN {X 0,Y 254.364,Z 722.911,A -85,B 0,C 180,E1 -18650.045,E2 -18650.045} C_VEL
LIN {X 0,Y 254.779,Z 721.877,A -85,B 0,C 180,E1 -18652.715,E2 -18652.715} C_VEL
LIN {X 0,Y 255.801,Z 719.566,A -85,B 0,C 180,E1 -18656.076,E2 -18656.076} C_VEL
LIN {X 0,Y 257.301,Z 716.192,A -85,B 0,C 180,E1 -18659.447,E2 -18659.447} C_VEL
LIN {X 0,Y 259.316,Z 711.526,A -85,B 0,C 180,E1 -18662.841,E2 -18662.841} C_VEL
LIN {X 0,Y 262.379,Z 704.877,A -85,B 0,C 180,E1 -18666.526,E2 -18666.526} C_VEL
LIN {X 0,Y 265.468,Z 698.234,A -85,B 0,C 180,E1 -18669.445,E2 -18669.445} C_VEL
LIN {X 0,Y 269.678,Z 689.206,A -85,B 0,C 180,E1 -18672.652,E2 -18672.652} C_VEL
LIN {X 0,Y 273.939,Z 679.757,A -85,B 0,C 180,E1 -18675.39,E2 -18675.39} C_VEL
LIN {X 0,Y 277.974,Z 670.159,A -85,B 0,C 180,E1 -18677.688,E2 -18677.688} C_VEL
LIN {X 0,Y 282.76,Z 658.294,A -85,B 0,C 180,E1 -18680.048,E2 -18680.048} C_VEL
LIN {X 0,Y 287.341,Z 645.858,A -85,B 0,C 180,E1 -18682.094,E2 -18682.094} C_VEL
LIN {X 0,Y 291.633,Z 633.046,A -85,B 0,C 180,E1 -18683.83,E2 -18683.83} C_VEL
LIN {X 0,Y 295.675,Z 619.066,A -85,B 0,C 180,E1 -18685.39,E2 -18685.39} C_VEL
LIN {X 0,Y 297.037,Z 613.835,A -85,B 0,C 180,E1 -18685.902,E2 -18685.902} C_VEL
LIN {X 0,Y 295.515,Z 605.052,A -85,B 0,C 180,E1 -18687.471,E2 -18687.471} C_VEL
LIN {X 0,Y 292.381,Z 593.392,A -85,B 0,C 180,E1 -18689.682,E2 -18689.682} C_VEL
LIN {X 0,Y 288.426,Z 583.16,A -85,B 0,C 180,E1 -18691.828,E2 -18691.828} C_VEL
LIN {X 0,Y 283.941,Z 574.393,A -85,B 0,C 180,E1 -18693.937,E2 -18693.937} C_VEL
LIN {X 0,Y 278.808,Z 565.736,A -85,B 0,C 180,E1 -18696.263,E2 -18696.263} C_VEL
LIN {X 0,Y 275.706,Z 561.079,A -85,B 0,C 180,E1 -18697.667,E2 -18697.667} C_VEL
LIN {X 0,Y 272.508,Z 556.478,A -85,B 0,C 180,E1 -18699.131,E2 -18699.131} C_VEL
LIN {X 0,Y 269.716,Z 552.786,A -85,B 0,C 180,E1 -18700.447,E2 -18700.447} C_VEL
LIN {X 0,Y 268.744,Z 551.408,A -85,B 0,C 180,E1 -18700.931,E2 -18700.931} C_VEL
LIN {X 0,Y 265.928,Z 548.177,A -85,B 0,C 180,E1 -18702.299,E2 -18702.299} C_VEL
LIN {X 0,Y 264.727,Z 546.293,A -85,B 0,C 180,E1 -18702.94,E2 -18702.94} C_VEL
LIN {X 0,Y 261.758,Z 543.292,A -85,B 0,C 180,E1 -18704.524,E2 -18704.524} C_VEL
LIN {X 0,Y 260.281,Z 540.703,A -85,B 0,C 180,E1 -18705.536,E2 -18705.536} C_VEL
LIN {X 0,Y 259.684,Z 537.401,A -85,B 0,C 180,E1 -18710.803,E2 -18710.803} C_VEL
LIN {X 0,Y 259.311,Z 535.846,A -85,B 0,C 180,E1 -18713.776,E2 -18713.776} C_VEL
LIN {X 0,Y 259.01,Z 534.231,A -85,B 0,C 180,E1 -18717.498,E2 -18717.498} C_VEL
LIN {X 0,Y 258.394,Z 534.134,A -85,B 0,C 180,E1 -18718.797,E2 -18718.797} C_VEL
LIN {X 0,Y 255.823,Z 535.089,A -85,B 0,C 180,E1 -18720.921,E2 -18720.921} C_VEL
LIN {X 0,Y 253.622,Z 536.102,A -85,B 0,C 180,E1 -18722.648,E2 -18722.648} C_VEL
LIN {X 0,Y 252.645,Z 536.556,A -85,B 0,C 180,E1 -18723.983,E2 -18723.983} C_VEL
LIN {X 0,Y 252.548,Z 536.591,A -85,B 0,C 180,E1 -18724.436,E2 -18724.436} C_VEL
LIN {X 0,Y 252.682,Z 536.515,A -85,B 0,C 180,E1 -18727.993,E2 -18727.993} C_VEL
LIN {X 0,Y 253.041,Z 537.421,A -85,B 0,C 180,E1 -18732.837,E2 -18732.837} C_VEL
LIN {X 0,Y 253.577,Z 538.64,A -85,B 0,C 180,E1 -18736.09,E2 -18736.09} C_VEL
LIN {X 0,Y 254.858,Z 541.57,A -85,B 0,C 180,E1 -18741.007,E2 -18741.007} C_VEL
LIN {X 0,Y 256.62,Z 545.292,A -85,B 0,C 180,E1 -18745.348,E2 -18745.348} C_VEL
LIN {X 0,Y 257.705,Z 547.854,A -85,B 0,C 180,E1 -18747.62,E2 -18747.62} C_VEL
LIN {X 0,Y 258.228,Z 550.263,A -85,B 0,C 180,E1 -18749.124,E2 -18749.124} C_VEL
LIN {X 0,Y 261.637,Z 555.894,A -85,B 0,C 180,E1 -18751.203,E2 -18751.203} C_VEL
LIN {X 0,Y 266.489,Z 563.669,A -85,B 0,C 180,E1 -18753.799,E2 -18753.799} C_VEL
LIN {X 0,Y 270.576,Z 570.997,A -85,B 0,C 180,E1 -18755.819,E2 -18755.819} C_VEL
LIN {X 0,Y 275.313,Z 579.431,A -85,B 0,C 180,E1 -18758.006,E2 -18758.006} C_VEL
LIN {X 0,Y 279.592,Z 588.818,A -85,B 0,C 180,E1 -18760.041,E2 -18760.041} C_VEL
LIN {X 0,Y 282.145,Z 595.96,A -85,B 0,C 180,E1 -18761.376,E2 -18761.376} C_VEL
LIN {X 0,Y 284.165,Z 608.183,A -85,B 0,C 180,E1 -18763.1,E2 -18763.1} C_VEL
LIN {X 0,Y 285.617,Z 623.494,A -85,B 0,C 180,E1 -18765.218,E2 -18765.218} C_VEL
LIN {X 0,Y 285.513,Z 638.778,A -85,B 0,C 180,E1 -18767.285,E2 -18767.285} C_VEL
LIN {X 0,Y 284.802,Z 651.726,A -85,B 0,C 180,E1 -18769.164,E2 -18769.164} C_VEL
LIN {X 0,Y 279.954,Z 666.365,A -85,B 0,C 180,E1 -18770.898,E2 -18770.898} C_VEL
LIN {X 0,Y 275.464,Z 678.666,A -85,B 0,C 180,E1 -18772.706,E2 -18772.706} C_VEL
LIN {X 0,Y 270.918,Z 690.294,A -85,B 0,C 180,E1 -18774.749,E2 -18774.749} C_VEL
LIN {X 0,Y 266.162,Z 701.974,A -85,B 0,C 180,E1 -18777.23,E2 -18777.23} C_VEL
LIN {X 0,Y 261.39,Z 713.274,A -85,B 0,C 180,E1 -18780.174,E2 -18780.174} C_VEL
LIN {X 0,Y 257.224,Z 722.775,A -85,B 0,C 180,E1 -18783.206,E2 -18783.206} C_VEL
LIN {X 0,Y 253.843,Z 730.929,A -85,B 0,C 180,E1 -18786.395,E2 -18786.395} C_VEL
LIN {X 0,Y 251.298,Z 737.554,A -85,B 0,C 180,E1 -18789.54,E2 -18789.54} C_VEL
LIN {X 0,Y 249.029,Z 744.297,A -85,B 0,C 180,E1 -18793.609,E2 -18793.609} C_VEL
LIN {X 0,Y 247.856,Z 748.426,A -85,B 0,C 180,E1 -18796.891,E2 -18796.891} C_VEL
LIN {X 0,Y 247.252,Z 751.58,A -85,B 0,C 180,E1 -18800.182,E2 -18800.182} C_VEL
LIN {X 0,Y 247.249,Z 754.072,A -85,B 0,C 180,E1 -18804.186,E2 -18804.186} C_VEL
LIN {X 0,Y 247.22,Z 754.855,A -85,B 0,C 180,E1 -18806.742,E2 -18806.742} C_VEL
LIN {X 0,Y 247.392,Z 754.982,A -85,B 0,C 180,E1 -18810.002,E2 -18810.002} C_VEL
LIN {X 0,Y 247.264,Z 754.11,A -85,B 0,C 180,E1 -18813.26,E2 -18813.26} C_VEL
LIN {X 0,Y 247.257,Z 752.179,A -85,B 0,C 180,E1 -18816.53,E2 -18816.53} C_VEL
LIN {X 0,Y 247.324,Z 749.185,A -85,B 0,C 180,E1 -18819.818,E2 -18819.818} C_VEL
LIN {X 0,Y 247.905,Z 745.111,A -85,B 0,C 180,E1 -18823.11,E2 -18823.11} C_VEL
LIN {X 0,Y 248.94,Z 739.823,A -85,B 0,C 180,E1 -18826.4,E2 -18826.4} C_VEL
LIN {X 0,Y 250.584,Z 733.335,A -85,B 0,C 180,E1 -18829.669,E2 -18829.669} C_VEL
LIN {X 0,Y 252.876,Z 725.811,A -85,B 0,C 180,E1 -18832.9,E2 -18832.9} C_VEL
LIN {X 0,Y 256.875,Z 716.777,A -85,B 0,C 180,E1 -18836.837,E2 -18836.837} C_VEL
LIN {X 0,Y 262.298,Z 706.298,A -85,B 0,C 180,E1 -18840.604,E2 -18840.604} C_VEL
LIN {X 0,Y 268.965,Z 694.36,A -85,B 0,C 180,E1 -18844.181,E2 -18844.181} C_VEL
LIN {X 0,Y 275.303,Z 683.722,A -85,B 0,C 180,E1 -18846.865,E2 -18846.865} C_VEL
LIN {X 0,Y 283.591,Z 670.503,A -85,B 0,C 180,E1 -18849.683,E2 -18849.683} C_VEL
LIN {X 0,Y 291.8,Z 657.928,A -85,B 0,C 180,E1 -18851.942,E2 -18851.942} C_VEL
LIN {X 0,Y 303.126,Z 638.684,A -85,B 0,C 180,E1 -18855.952,E2 -18855.952} C_VEL
LIN {X 0,Y 307.337,Z 632.157,A -85,B 0,C 180,E1 -18857.566,E2 -18857.566} C_VEL
LIN {X 0,Y 309.556,Z 629.069,A -85,B 0,C 180,E1 -18858.524,E2 -18858.524} C_VEL
LIN {X 0,Y 309.024,Z 629.708,A -85,B 0,C 180,E1 -18858.736,E2 -18858.736} C_VEL
LIN {X 0,Y 298.09,Z 643.254,A -85,B 0,C 180,E1 -18861.334,E2 -18861.334} C_VEL
LIN {X 0,Y 288.275,Z 655.153,A -85,B 0,C 180,E1 -18864.19,E2 -18864.19} C_VEL
LIN {X 0,Y 279.695,Z 665.49,A -85,B 0,C 180,E1 -18867.301,E2 -18867.301} C_VEL
LIN {X 0,Y 272.162,Z 674.352,A -85,B 0,C 180,E1 -18870.619,E2 -18870.619} C_VEL
LIN {X 0,Y 265.546,Z 682.097,A -85,B 0,C 180,E1 -18874.298,E2 -18874.298} C_VEL
LIN {X 0,Y 260.542,Z 687.836,A -85,B 0,C 180,E1 -18877.813,E2 -18877.813} C_VEL
LIN {X 0,Y 257.089,Z 691.621,A -85,B 0,C 180,E1 -18880.851,E2 -18880.851} C_VEL
LIN {X 0,Y 254.261,Z 694.578,A -85,B 0,C 180,E1 -18883.955,E2 -18883.955} C_VEL
LIN {X 0,Y 251.859,Z 696.888,A -85,B 0,C 180,E1 -18887.601,E2 -18887.601} C_VEL
LIN {X 0,Y 249.975,Z 698.075,A -85,B 0,C 180,E1 -18891.92,E2 -18891.92} C_VEL
LIN {X 0,Y 248.896,Z 697.895,A -85,B 0,C 180,E1 -18895.141,E2 -18895.141} C_VEL
LIN {X 0,Y 248.263,Z 696.858,A -85,B 0,C 180,E1 -18898.379,E2 -18898.379} C_VEL
LIN {X 0,Y 248.158,Z 694.803,A -85,B 0,C 180,E1 -18901.624,E2 -18901.624} C_VEL
LIN {X 0,Y 248.392,Z 691.798,A -85,B 0,C 180,E1 -18904.87,E2 -18904.87} C_VEL
LIN {X 0,Y 248.71,Z 687.274,A -85,B 0,C 180,E1 -18908.491,E2 -18908.491} C_VEL
LIN {X 0,Y 249.46,Z 681.197,A -85,B 0,C 180,E1 -18912.199,E2 -18912.199} C_VEL
LIN {X 0,Y 250.585,Z 674.525,A -85,B 0,C 180,E1 -18915.453,E2 -18915.453} C_VEL
LIN {X 0,Y 252.249,Z 666.536,A -85,B 0,C 180,E1 -18918.683,E2 -18918.683} C_VEL
LIN {X 0,Y 254.487,Z 656.998,A -85,B 0,C 180,E1 -18921.89,E2 -18921.89} C_VEL
LIN {X 0,Y 257.254,Z 645.71,A -85,B 0,C 180,E1 -18925.053,E2 -18925.053} C_VEL
LIN {X 0,Y 260.051,Z 634.147,A -85,B 0,C 180,E1 -18927.788,E2 -18927.788} C_VEL
LIN {X 0,Y 263.437,Z 620.65,A -85,B 0,C 180,E1 -18930.457,E2 -18930.457} C_VEL
LIN {X 0,Y 266.918,Z 606.067,A -85,B 0,C 180,E1 -18932.868,E2 -18932.868} C_VEL
LIN {X 0,Y 270.389,Z 590.142,A -85,B 0,C 180,E1 -18935.057,E2 -18935.057} C_VEL
LIN {X 0,Y 271.892,Z 582.953,A -85,B 0,C 180,E1 -18935.911,E2 -18935.911} C_VEL
LIN {X 0,Y 267.064,Z 569.48,A -85,B 0,C 180,E1 -18938.168,E2 -18938.168} C_VEL
LIN {X 0,Y 261.018,Z 554.056,A -85,B 0,C 180,E1 -18940.652,E2 -18940.652} C_VEL
LIN {X 0,Y 254.4,Z 539.571,A -85,B 0,C 180,E1 -18942.937,E2 -18942.937} C_VEL
LIN {X 0,Y 249.698,Z 530.007,A -85,B 0,C 180,E1 -18944.422,E2 -18944.422} C_VEL
LIN {X 0,Y 249.027,Z 527.778,A -85,B 0,C 180,E1 -18944.734,E2 -18944.734} C_VEL
LIN {X 0,Y 249.055,Z 527.842,A -85,B 0,C 180,E1 -18946.663,E2 -18946.663} C_VEL
LIN {X 0,Y 250.119,Z 532.298,A -85,B 0,C 180,E1 -18950.785,E2 -18950.785} C_VEL
LIN {X 0,Y 251.193,Z 537.227,A -85,B 0,C 180,E1 -18955.176,E2 -18955.176} C_VEL
LIN {X 0,Y 252.835,Z 540.524,A -85,B 0,C 180,E1 -18955.69,E2 -18955.69} C_VEL
LIN {X 0,Y 254.601,Z 542.846,A -85,B 0,C 180,E1 -18956.17,E2 -18956.17} C_VEL
LIN {X 0,Y 260.149,Z 552.032,A -85,B 0,C 180,E1 -18957.734,E2 -18957.734} C_VEL
LIN {X 0,Y 265.69,Z 562.179,A -85,B 0,C 180,E1 -18959.376,E2 -18959.376} C_VEL
LIN {X 0,Y 270.258,Z 572.89,A -85,B 0,C 180,E1 -18960.937,E2 -18960.937} C_VEL
LIN {X 0,Y 274.578,Z 586.086,A -85,B 0,C 180,E1 -18962.805,E2 -18962.805} C_VEL
LIN {X 0,Y 278.343,Z 600.228,A -85,B 0,C 180,E1 -18964.851,E2 -18964.851} C_VEL
LIN {X 0,Y 279.81,Z 607.37,A -85,B 0,C 180,E1 -18965.905,E2 -18965.905} C_VEL
LIN {X 0,Y 276.847,Z 621.806,A -85,B 0,C 180,E1 -18967.419,E2 -18967.419} C_VEL
LIN {X 0,Y 273.454,Z 635.29,A -85,B 0,C 180,E1 -18969.107,E2 -18969.107} C_VEL
LIN {X 0,Y 269.557,Z 648.988,A -85,B 0,C 180,E1 -18971.176,E2 -18971.176} C_VEL
LIN {X 0,Y 265.782,Z 661.523,A -85,B 0,C 180,E1 -18973.484,E2 -18973.484} C_VEL
LIN {X 0,Y 262.103,Z 673.02,A -85,B 0,C 180,E1 -18976.034,E2 -18976.034} C_VEL
LIN {X 0,Y 258.808,Z 682.766,A -85,B 0,C 180,E1 -18978.644,E2 -18978.644} C_VEL
LIN {X 0,Y 255.777,Z 691.873,A -85,B 0,C 180,E1 -18981.567,E2 -18981.567} C_VEL
LIN {X 0,Y 253.214,Z 699.363,A -85,B 0,C 180,E1 -18984.424,E2 -18984.424} C_VEL
LIN {X 0,Y 251.088,Z 706.102,A -85,B 0,C 180,E1 -18987.592,E2 -18987.592} C_VEL
LIN {X 0,Y 249.407,Z 711.664,A -85,B 0,C 180,E1 -18990.806,E2 -18990.806} C_VEL
LIN {X 0,Y 248.592,Z 715.085,A -85,B 0,C 180,E1 -18993.24,E2 -18993.24} C_VEL
LIN {X 0,Y 247.681,Z 718.95,A -85,B 0,C 180,E1 -18996.713,E2 -18996.713} C_VEL
LIN {X 0,Y 247.202,Z 721.405,A -85,B 0,C 180,E1 -18999.82,E2 -18999.82} C_VEL
LIN {X 0,Y 246.988,Z 723.076,A -85,B 0,C 180,E1 -19003.156,E2 -19003.156} C_VEL
LIN {X 0,Y 246.958,Z 723.782,A -85,B 0,C 180,E1 -19006.532,E2 -19006.532} C_VEL
LIN {X 0,Y 247.314,Z 723.369,A -85,B 0,C 180,E1 -19010.317,E2 -19010.317} C_VEL
LIN {X 0,Y 247.855,Z 722.191,A -85,B 0,C 180,E1 -19013.387,E2 -19013.387} C_VEL
LIN {X 0,Y 249,Z 719.759,A -85,B 0,C 180,E1 -19016.844,E2 -19016.844} C_VEL
LIN {X 0,Y 250.672,Z 716.253,A -85,B 0,C 180,E1 -19020.306,E2 -19020.306} C_VEL
LIN {X 0,Y 252.891,Z 711.547,A -85,B 0,C 180,E1 -19023.764,E2 -19023.764} C_VEL
LIN {X 0,Y 255.868,Z 705.418,A -85,B 0,C 180,E1 -19027.197,E2 -19027.197} C_VEL
LIN {X 0,Y 259.549,Z 697.925,A -85,B 0,C 180,E1 -19030.529,E2 -19030.529} C_VEL
LIN {X 0,Y 264.031,Z 688.73,A -85,B 0,C 180,E1 -19033.791,E2 -19033.791} C_VEL
LIN {X 0,Y 268.571,Z 679.1,A -85,B 0,C 180,E1 -19036.563,E2 -19036.563} C_VEL
LIN {X 0,Y 272.879,Z 669.385,A -85,B 0,C 180,E1 -19038.877,E2 -19038.877} C_VEL
LIN {X 0,Y 277.674,Z 657.813,A -85,B 0,C 180,E1 -19041.163,E2 -19041.163} C_VEL
LIN {X 0,Y 282.386,Z 645.445,A -85,B 0,C 180,E1 -19043.186,E2 -19043.186} C_VEL
LIN {X 0,Y 286.726,Z 632.906,A -85,B 0,C 180,E1 -19044.887,E2 -19044.887} C_VEL
LIN {X 0,Y 290.779,Z 619.312,A -85,B 0,C 180,E1 -19046.406,E2 -19046.406} C_VEL
LIN {X 0,Y 291.644,Z 615.974,A -85,B 0,C 180,E1 -19046.754,E2 -19046.754} C_VEL
LIN {X 0,Y 289.894,Z 606.347,A -85,B 0,C 180,E1 -19048.584,E2 -19048.584} C_VEL
LIN {X 0,Y 287.126,Z 595.826,A -85,B 0,C 180,E1 -19050.689,E2 -19050.689} C_VEL
LIN {X 0,Y 283.656,Z 586.791,A -85,B 0,C 180,E1 -19052.718,E2 -19052.718} C_VEL
LIN {X 0,Y 279.542,Z 578.579,A -85,B 0,C 180,E1 -19054.829,E2 -19054.829} C_VEL
LIN {X 0,Y 275.475,Z 571.347,A -85,B 0,C 180,E1 -19056.855,E2 -19056.855} C_VEL
LIN {X 0,Y 272.658,Z 566.895,A -85,B 0,C 180,E1 -19058.251,E2 -19058.251} C_VEL
LIN {X 0,Y 269.785,Z 562.547,A -85,B 0,C 180,E1 -19059.689,E2 -19059.689} C_VEL
LIN {X 0,Y 266.924,Z 558.365,A -85,B 0,C 180,E1 -19061.17,E2 -19061.17} C_VEL
LIN {X 0,Y 263.471,Z 554.085,A -85,B 0,C 180,E1 -19062.979,E2 -19062.979} C_VEL
LIN {X 0,Y 262.459,Z 552.535,A -85,B 0,C 180,E1 -19063.57,E2 -19063.57} C_VEL
LIN {X 0,Y 259.576,Z 549.353,A -85,B 0,C 180,E1 -19065.195,E2 -19065.195} C_VEL
LIN {X 0,Y 258.079,Z 547.133,A -85,B 0,C 180,E1 -19066.133,E2 -19066.133} C_VEL
LIN {X 0,Y 254.865,Z 544.002,A -85,B 0,C 180,E1 -19068.215,E2 -19068.215} C_VEL
LIN {X 0,Y 253.581,Z 541.743,A -85,B 0,C 180,E1 -19069.217,E2 -19069.217} C_VEL
LIN {X 0,Y 253.371,Z 540.208,A -85,B 0,C 180,E1 -19072.027,E2 -19072.027} C_VEL
LIN {X 0,Y 252.94,Z 537.905,A -85,B 0,C 180,E1 -19077.564,E2 -19077.564} C_VEL
LIN {X 0,Y 252.96,Z 537.143,A -85,B 0,C 180,E1 -19079.999,E2 -19079.999} C_VEL
LIN {X 0,Y 252.682,Z 536.597,A -85,B 0,C 180,E1 -19083.188,E2 -19083.188} C_VEL
LIN {X 0,Y 252.548,Z 536.591,A -85,B 0,C 180,E1 -19084.436,E2 -19084.436} C_VEL
LIN {X 0,Y 251.961,Z 536.968,A -85,B 0,C 180,E1 -19085.768,E2 -19085.768} C_VEL
LIN {X 0,Y 249.677,Z 538.671,A -85,B 0,C 180,E1 -19087.937,E2 -19087.937} C_VEL
LIN {X 0,Y 247.825,Z 540.25,A -85,B 0,C 180,E1 -19089.694,E2 -19089.694} C_VEL
LIN {X 0,Y 247.118,Z 541.118,A -85,B 0,C 180,E1 -19091.052,E2 -19091.052} C_VEL
LIN {X 0,Y 247.104,Z 541.289,A -85,B 0,C 180,E1 -19091.512,E2 -19091.512} C_VEL
LIN {X 0,Y 247.784,Z 542.641,A -85,B 0,C 180,E1 -19095.352,E2 -19095.352} C_VEL
LIN {X 0,Y 248.887,Z 545.157,A -85,B 0,C 180,E1 -19099.806,E2 -19099.806} C_VEL
LIN {X 0,Y 250.194,Z 547.799,A -85,B 0,C 180,E1 -19103.157,E2 -19103.157} C_VEL
LIN {X 0,Y 251.023,Z 549.441,A -85,B 0,C 180,E1 -19104.721,E2 -19104.721} C_VEL
LIN {X 0,Y 256.132,Z 556.313,A -85,B 0,C 180,E1 -19108.438,E2 -19108.438} C_VEL
LIN {X 0,Y 259.46,Z 562.023,A -85,B 0,C 180,E1 -19110.571,E2 -19110.571} C_VEL
LIN {X 0,Y 264.137,Z 569.91,A -85,B 0,C 180,E1 -19113.225,E2 -19113.225} C_VEL
LIN {X 0,Y 268.336,Z 577.802,A -85,B 0,C 180,E1 -19115.451,E2 -19115.451} C_VEL
LIN {X 0,Y 271.981,Z 584.84,A -85,B 0,C 180,E1 -19117.323,E2 -19117.323} C_VEL
LIN {X 0,Y 275.768,Z 593.792,A -85,B 0,C 180,E1 -19119.341,E2 -19119.341} C_VEL
LIN {X 0,Y 277.891,Z 600.173,A -85,B 0,C 180,E1 -19120.596,E2 -19120.596} C_VEL
LIN {X 0,Y 279.644,Z 613.399,A -85,B 0,C 180,E1 -19122.527,E2 -19122.527} C_VEL
LIN {X 0,Y 280.539,Z 627.312,A -85,B 0,C 180,E1 -19124.543,E2 -19124.543} C_VEL
LIN {X 0,Y 280.071,Z 642.559,A -85,B 0,C 180,E1 -19126.694,E2 -19126.694} C_VEL
LIN {X 0,Y 279.368,Z 652.358,A -85,B 0,C 180,E1 -19128.197,E2 -19128.197} C_VEL
LIN {X 0,Y 274.935,Z 665.58,A -85,B 0,C 180,E1 -19129.803,E2 -19129.803} C_VEL
LIN {X 0,Y 269.846,Z 678.966,A -85,B 0,C 180,E1 -19131.792,E2 -19131.792} C_VEL
LIN {X 0,Y 265.128,Z 690.465,A -85,B 0,C 180,E1 -19133.86,E2 -19133.86} C_VEL
LIN {X 0,Y 260.174,Z 702.039,A -85,B 0,C 180,E1 -19136.377,E2 -19136.377} C_VEL
LIN {X 0,Y 256.342,Z 710.59,A -85,B 0,C 180,E1 -19138.609,E2 -19138.609} C_VEL
LIN {X 0,Y 251.814,Z 720.452,A -85,B 0,C 180,E1 -19141.678,E2 -19141.678} C_VEL
LIN {X 0,Y 248.127,Z 728.806,A -85,B 0,C 180,E1 -19144.86,E2 -19144.86} C_VEL
LIN {X 0,Y 245.191,Z 735.768,A -85,B 0,C 180,E1 -19148.125,E2 -19148.125} C_VEL
LIN {X 0,Y 242.946,Z 741.524,A -85,B 0,C 180,E1 -19151.447,E2 -19151.447} C_VEL
LIN {X 0,Y 241.44,Z 746.214,A -85,B 0,C 180,E1 -19154.815,E2 -19154.815} C_VEL
LIN {X 0,Y 240.407,Z 749.769,A -85,B 0,C 180,E1 -19158.194,E2 -19158.194} C_VEL
LIN {X 0,Y 240.054,Z 752.405,A -85,B 0,C 180,E1 -19161.585,E2 -19161.585} C_VEL
LIN {X 0,Y 240.113,Z 753.968,A -85,B 0,C 180,E1 -19164.964,E2 -19164.964} C_VEL
LIN {X 0,Y 240.176,Z 754.62,A -85,B 0,C 180,E1 -19168.325,E2 -19168.325} C_VEL
LIN {X 0,Y 240.304,Z 754.518,A -85,B 0,C 180,E1 -19170.002,E2 -19170.002} C_VEL
LIN {X 0,Y 240.195,Z 753.597,A -85,B 0,C 180,E1 -19173.357,E2 -19173.357} C_VEL
LIN {X 0,Y 240.172,Z 751.639,A -85,B 0,C 180,E1 -19176.724,E2 -19176.724} C_VEL
LIN {X 0,Y 240.272,Z 748.592,A -85,B 0,C 180,E1 -19180.109,E2 -19180.109} C_VEL
LIN {X 0,Y 240.904,Z 744.49,A -85,B 0,C 180,E1 -19183.498,E2 -19183.498} C_VEL
LIN {X 0,Y 242.022,Z 739.144,A -85,B 0,C 180,E1 -19186.883,E2 -19186.883} C_VEL
LIN {X 0,Y 243.774,Z 732.595,A -85,B 0,C 180,E1 -19190.242,E2 -19190.242} C_VEL
LIN {X 0,Y 244.916,Z 728.844,A -85,B 0,C 180,E1 -19191.905,E2 -19191.905} C_VEL
LIN {X 0,Y 248.637,Z 720.658,A -85,B 0,C 180,E1 -19195.986,E2 -19195.986} C_VEL
LIN {X 0,Y 253.76,Z 711.133,A -85,B 0,C 180,E1 -19199.904,E2 -19199.904} C_VEL
LIN {X 0,Y 260.959,Z 699.061,A -85,B 0,C 180,E1 -19203.976,E2 -19203.976} C_VEL
LIN {X 0,Y 268.929,Z 686.693,A -85,B 0,C 180,E1 -19207.418,E2 -19207.418} C_VEL
LIN {X 0,Y 277.452,Z 674.141,A -85,B 0,C 180,E1 -19210.295,E2 -19210.295} C_VEL
LIN {X 0,Y 287.92,Z 659.322,A -85,B 0,C 180,E1 -19213.117,E2 -19213.117} C_VEL
LIN {X 0,Y 299.023,Z 642.647,A -85,B 0,C 180,E1 -19216.77,E2 -19216.77} C_VEL
LIN {X 0,Y 302.621,Z 637.685,A -85,B 0,C 180,E1 -19218.003,E2 -19218.003} C_VEL
LIN {X 0,Y 303.129,Z 637.002,A -85,B 0,C 180,E1 -19218.378,E2 -19218.378} C_VEL
LIN {X 0,Y 291.303,Z 650.166,A -85,B 0,C 180,E1 -19221.151,E2 -19221.151} C_VEL
LIN {X 0,Y 280.448,Z 662.049,A -85,B 0,C 180,E1 -19224.364,E2 -19224.364} C_VEL
LIN {X 0,Y 271.059,Z 672.21,A -85,B 0,C 180,E1 -19227.892,E2 -19227.892} C_VEL
LIN {X 0,Y 263.651,Z 680.04,A -85,B 0,C 180,E1 -19231.327,E2 -19231.327} C_VEL
LIN {X 0,Y 257.417,Z 686.543,A -85,B 0,C 180,E1 -19234.965,E2 -19234.965} C_VEL
LIN {X 0,Y 252.324,Z 691.696,A -85,B 0,C 180,E1 -19238.772,E2 -19238.772} C_VEL
LIN {X 0,Y 248.999,Z 694.82,A -85,B 0,C 180,E1 -19241.913,E2 -19241.913} C_VEL
LIN {X 0,Y 246.349,Z 697.147,A -85,B 0,C 180,E1 -19245.123,E2 -19245.123} C_VEL
LIN {X 0,Y 244.386,Z 698.553,A -85,B 0,C 180,E1 -19248.388,E2 -19248.388} C_VEL
LIN {X 0,Y 243.032,Z 699.112,A -85,B 0,C 180,E1 -19251.687,E2 -19251.687} C_VEL
LIN {X 0,Y 241.892,Z 698.825,A -85,B 0,C 180,E1 -19255,E2 -19255} C_VEL
LIN {X 0,Y 241.229,Z 697.597,A -85,B 0,C 180,E1 -19258.331,E2 -19258.331} C_VEL
LIN {X 0,Y 241.096,Z 695.437,A -85,B 0,C 180,E1 -19261.671,E2 -19261.671} C_VEL
LIN {X 0,Y 241.312,Z 692.262,A -85,B 0,C 180,E1 -19265.013,E2 -19265.013} C_VEL
LIN {X 0,Y 241.643,Z 687.854,A -85,B 0,C 180,E1 -19268.552,E2 -19268.552} C_VEL
LIN {X 0,Y 242.474,Z 681.329,A -85,B 0,C 180,E1 -19272.556,E2 -19272.556} C_VEL
LIN {X 0,Y 243.691,Z 674.512,A -85,B 0,C 180,E1 -19275.902,E2 -19275.902} C_VEL
LIN {X 0,Y 245.542,Z 666.065,A -85,B 0,C 180,E1 -19279.318,E2 -19279.318} C_VEL
LIN {X 0,Y 247.798,Z 656.599,A -85,B 0,C 180,E1 -19282.513,E2 -19282.513} C_VEL
LIN {X 0,Y 250.649,Z 645.202,A -85,B 0,C 180,E1 -19285.736,E2 -19285.736} C_VEL
LIN {X 0,Y 253.642,Z 633.298,A -85,B 0,C 180,E1 -19288.554,E2 -19288.554} C_VEL
LIN {X 0,Y 257.201,Z 619.51,A -85,B 0,C 180,E1 -19291.278,E2 -19291.278} C_VEL
LIN {X 0,Y 260.571,Z 605.724,A -85,B 0,C 180,E1 -19293.567,E2 -19293.567} C_VEL
LIN {X 0,Y 263.867,Z 590.949,A -85,B 0,C 180,E1 -19295.637,E2 -19295.637} C_VEL
LIN {X 0,Y 265.165,Z 585.06,A -85,B 0,C 180,E1 -19296.348,E2 -19296.348} C_VEL
LIN {X 0,Y 260.754,Z 572.225,A -85,B 0,C 180,E1 -19298.589,E2 -19298.589} C_VEL
LIN {X 0,Y 255.573,Z 558.691,A -85,B 0,C 180,E1 -19300.866,E2 -19300.866} C_VEL
LIN {X 0,Y 248.876,Z 543.6,A -85,B 0,C 180,E1 -19303.35,E2 -19303.35} C_VEL
LIN {X 0,Y 243.017,Z 531.576,A -85,B 0,C 180,E1 -19305.321,E2 -19305.321} C_VEL
LIN {X 0,Y 242.115,Z 529.447,A -85,B 0,C 180,E1 -19305.693,E2 -19305.693} C_VEL
LIN {X 0,Y 242.961,Z 532.601,A -85,B 0,C 180,E1 -19308.773,E2 -19308.773} C_VEL
LIN {X 0,Y 244.1,Z 537.615,A -85,B 0,C 180,E1 -19313.438,E2 -19313.438} C_VEL
LIN {X 0,Y 244.287,Z 538.194,A -85,B 0,C 180,E1 -19313.593,E2 -19313.593} C_VEL
LIN {X 0,Y 246.333,Z 541.634,A -85,B 0,C 180,E1 -19314.234,E2 -19314.234} C_VEL
LIN {X 0,Y 247.719,Z 543.602,A -85,B 0,C 180,E1 -19314.645,E2 -19314.645} C_VEL
LIN {X 0,Y 253.247,Z 552.29,A -85,B 0,C 180,E1 -19316.296,E2 -19316.296} C_VEL
LIN {X 0,Y 260.216,Z 565.007,A -85,B 0,C 180,E1 -19318.481,E2 -19318.481} C_VEL
LIN {X 0,Y 264.774,Z 575.823,A -85,B 0,C 180,E1 -19320.175,E2 -19320.175} C_VEL
LIN {X 0,Y 268.514,Z 587.398,A -85,B 0,C 180,E1 -19321.891,E2 -19321.891} C_VEL
LIN {X 0,Y 272.038,Z 601.062,A -85,B 0,C 180,E1 -19323.947,E2 -19323.947} C_VEL
LIN {X 0,Y 273.732,Z 609.379,A -85,B 0,C 180,E1 -19325.237,E2 -19325.237} C_VEL
LIN {X 0,Y 270.429,Z 624.375,A -85,B 0,C 180,E1 -19326.853,E2 -19326.853} C_VEL
LIN {X 0,Y 266.574,Z 638.797,A -85,B 0,C 180,E1 -19328.744,E2 -19328.744} C_VEL
LIN {X 0,Y 262.595,Z 651.986,A -85,B 0,C 180,E1 -19330.86,E2 -19330.86} C_VEL
LIN {X 0,Y 259.058,Z 663.231,A -85,B 0,C 180,E1 -19333.042,E2 -19333.042} C_VEL
LIN {X 0,Y 255.282,Z 674.524,A -85,B 0,C 180,E1 -19335.653,E2 -19335.653} C_VEL
LIN {X 0,Y 251.884,Z 684.181,A -85,B 0,C 180,E1 -19338.328,E2 -19338.328} C_VEL
LIN {X 0,Y 248.881,Z 692.894,A -85,B 0,C 180,E1 -19341.248,E2 -19341.248} C_VEL
LIN {X 0,Y 246.184,Z 700.455,A -85,B 0,C 180,E1 -19344.264,E2 -19344.264} C_VEL
LIN {X 0,Y 244.008,Z 707.128,A -85,B 0,C 180,E1 -19347.522,E2 -19347.522} C_VEL
LIN {X 0,Y 242.307,Z 712.558,A -85,B 0,C 180,E1 -19350.829,E2 -19350.829} C_VEL
LIN {X 0,Y 241.465,Z 715.922,A -85,B 0,C 180,E1 -19353.335,E2 -19353.335} C_VEL
LIN {X 0,Y 240.602,Z 719.492,A -85,B 0,C 180,E1 -19356.708,E2 -19356.708} C_VEL
LIN {X 0,Y 240.08,Z 722.068,A -85,B 0,C 180,E1 -19360.114,E2 -19360.114} C_VEL
LIN {X 0,Y 239.881,Z 723.624,A -85,B 0,C 180,E1 -19363.553,E2 -19363.553} C_VEL
LIN {X 0,Y 239.894,Z 724.275,A -85,B 0,C 180,E1 -19367.033,E2 -19367.033} C_VEL
LIN {X 0,Y 240.28,Z 723.826,A -85,B 0,C 180,E1 -19370.611,E2 -19370.611} C_VEL
LIN {X 0,Y 240.976,Z 722.458,A -85,B 0,C 180,E1 -19374.096,E2 -19374.096} C_VEL
LIN {X 0,Y 242.238,Z 719.954,A -85,B 0,C 180,E1 -19377.656,E2 -19377.656} C_VEL
LIN {X 0,Y 244.085,Z 716.315,A -85,B 0,C 180,E1 -19381.214,E2 -19381.214} C_VEL
LIN {X 0,Y 246.54,Z 711.501,A -85,B 0,C 180,E1 -19384.757,E2 -19384.757} C_VEL
LIN {X 0,Y 249.743,Z 705.314,A -85,B 0,C 180,E1 -19388.248,E2 -19388.248} C_VEL
LIN {X 0,Y 253.75,Z 697.63,A -85,B 0,C 180,E1 -19391.658,E2 -19391.658} C_VEL
LIN {X 0,Y 257.888,Z 689.536,A -85,B 0,C 180,E1 -19394.564,E2 -19394.564} C_VEL
LIN {X 0,Y 262.613,Z 679.977,A -85,B 0,C 180,E1 -19397.384,E2 -19397.384} C_VEL
LIN {X 0,Y 267.916,Z 668.619,A -85,B 0,C 180,E1 -19400.108,E2 -19400.108} C_VEL
LIN {X 0,Y 273.242,Z 656.119,A -85,B 0,C 180,E1 -19402.54,E2 -19402.54} C_VEL
LIN {X 0,Y 277.793,Z 644.376,A -85,B 0,C 180,E1 -19404.416,E2 -19404.416} C_VEL
LIN {X 0,Y 282.4,Z 631.252,A -85,B 0,C 180,E1 -19406.156,E2 -19406.156} C_VEL
LIN {X 0,Y 286.256,Z 618.613,A -85,B 0,C 180,E1 -19407.556,E2 -19407.556} C_VEL
LIN {X 0,Y 284.547,Z 608.521,A -85,B 0,C 180,E1 -19409.581,E2 -19409.581} C_VEL
LIN {X 0,Y 282.429,Z 599.95,A -85,B 0,C 180,E1 -19411.378,E2 -19411.378} C_VEL
LIN {X 0,Y 279.206,Z 591.144,A -85,B 0,C 180,E1 -19413.461,E2 -19413.461} C_VEL
LIN {X 0,Y 274.653,Z 581.589,A -85,B 0,C 180,E1 -19416.037,E2 -19416.037} C_VEL
LIN {X 0,Y 270.044,Z 573.343,A -85,B 0,C 180,E1 -19418.556,E2 -19418.556} C_VEL
LIN {X 0,Y 266.9,Z 568.46,A -85,B 0,C 180,E1 -19420.282,E2 -19420.282} C_VEL
LIN {X 0,Y 263.723,Z 563.765,A -85,B 0,C 180,E1 -19422.053,E2 -19422.053} C_VEL
LIN {X 0,Y 261.107,Z 560.182,A -85,B 0,C 180,E1 -19423.583,E2 -19423.583} C_VEL
LIN {X 0,Y 260.038,Z 558.688,A -85,B 0,C 180,E1 -19424.218,E2 -19424.218} C_VEL
LIN {X 0,Y 257.394,Z 555.445,A -85,B 0,C 180,E1 -19425.846,E2 -19425.846} C_VEL
LIN {X 0,Y 256.328,Z 553.765,A -85,B 0,C 180,E1 -19426.581,E2 -19426.581} C_VEL
LIN {X 0,Y 253.208,Z 550.574,A -85,B 0,C 180,E1 -19428.695,E2 -19428.695} C_VEL
LIN {X 0,Y 251.87,Z 548.398,A -85,B 0,C 180,E1 -19429.753,E2 -19429.753} C_VEL
LIN {X 0,Y 248.177,Z 544.795,A -85,B 0,C 180,E1 -19432.882,E2 -19432.882} C_VEL
LIN {X 0,Y 246.966,Z 542.766,A -85,B 0,C 180,E1 -19434.283,E2 -19434.283} C_VEL
LIN {X 0,Y 246.945,Z 541.389,A -85,B 0,C 180,E1 -19438.368,E2 -19438.368} C_VEL
LIN {X 0,Y 246.897,Z 540.639,A -85,B 0,C 180,E1 -19441.63,E2 -19441.63} C_VEL
LIN {X 0,Y 246.811,Z 540.526,A -85,B 0,C 180,E1 -19446.54,E2 -19446.54} C_VEL
LIN {X 0,Y 246.95,Z 540.914,A -85,B 0,C 180,E1 -19449.831,E2 -19449.831} C_VEL
LIN {X 0,Y 247.104,Z 541.289,A -85,B 0,C 180,E1 -19451.512,E2 -19451.512} C_VEL
